	VAR robtarget Openhole_6902 := [[456.45, -15.03, 181.27], [0.011887, 0.707007, 0.706156, -0.036651], [0,0,0,0], [9E9, 9E9, 9E9, 9E9, 9E9, 9E9]];
	VAR robtarget Openhole_6903 := [[454.01, -15.03, 181.36], [0.00355, 0.707098, 0.706536, -0.028396], [0,0,0,0], [9E9, 9E9, 9E9, 9E9, 9E9, 9E9]];
	VAR robtarget Openhole_6904 := [[454.58, -16.45, 181.41], [0.010332, 0.707031, 0.706647, -0.025509], [0,0,0,0], [9E9, 9E9, 9E9, 9E9, 9E9, 9E9]];
	VAR robtarget Openhole_6905 := [[457.02, -16.45, 181.35], [0.018656, 0.706861, 0.7063, -0.033765], [0,0,0,0], [9E9, 9E9, 9E9, 9E9, 9E9, 9E9]];
	VAR robtarget Openhole_6906 := [[457.6, -16.2, 181.32], [0.019746, 0.706831, 0.706161, -0.036559], [0,0,0,0], [9E9, 9E9, 9E9, 9E9, 9E9, 9E9]];
	VAR robtarget Openhole_6907 := [[458.49, -15.74, 181.25], [0.021192, 0.706789, 0.705912, -0.041085], [0,0,0,0], [9E9, 9E9, 9E9, 9E9, 9E9, 9E9]];
	VAR robtarget Openhole_6908 := [[458.92, -15.49, 181.22], [0.021819, 0.70677, 0.705775, -0.043372], [0,0,0,0], [9E9, 9E9, 9E9, 9E9, 9E9, 9E9]];
	VAR robtarget Openhole_6909 := [[459.34, -15.23, 181.18], [0.022372, 0.706753, 0.70563, -0.045673], [0,0,0,0], [9E9, 9E9, 9E9, 9E9, 9E9, 9E9]];
	VAR robtarget Openhole_6910 := [[460.18, -14.69, 181.09], [0.023376, 0.70672, 0.705316, -0.050289], [0,0,0,0], [9E9, 9E9, 9E9, 9E9, 9E9, 9E9]];
	VAR robtarget Openhole_6911 := [[461.04, -14.18, 181], [0.024553, 0.70668, 0.704976, -0.05485], [0,0,0,0], [9E9, 9E9, 9E9, 9E9, 9E9, 9E9]];
	VAR robtarget Openhole_6912 := [[463.23, -13.02, 180.74], [0.028061, 0.70655, 0.704018, -0.066023], [0,0,0,0], [9E9, 9E9, 9E9, 9E9, 9E9, 9E9]];
	VAR robtarget Openhole_6913 := [[463.68, -12.81, 180.68], [0.028865, 0.706517, 0.703809, -0.068211], [0,0,0,0], [9E9, 9E9, 9E9, 9E9, 9E9, 9E9]];
	VAR robtarget Openhole_6914 := [[465.05, -12.22, 180.51], [0.031491, 0.706405, 0.703154, -0.074666], [0,0,0,0], [9E9, 9E9, 9E9, 9E9, 9E9, 9E9]];
	VAR robtarget Openhole_6915 := [[465.52, -12.04, 180.45], [0.032438, 0.706362, 0.702926, -0.076778], [0,0,0,0], [9E9, 9E9, 9E9, 9E9, 9E9, 9E9]];
	VAR robtarget Openhole_6916 := [[468.83, -10.99, 180.03], [0.040018, 0.705973, 0.701231, -0.090969], [0,0,0,0], [9E9, 9E9, 9E9, 9E9, 9E9, 9E9]];
	VAR robtarget Openhole_6917 := [[469.79, -10.75, 179.91], [0.042431, 0.705833, 0.700718, -0.094841], [0,0,0,0], [9E9, 9E9, 9E9, 9E9, 9E9, 9E9]];
	VAR robtarget Openhole_6918 := [[473.7, -10.06, 179.44], [0.053059, 0.705113, 0.698584, -0.109453], [0,0,0,0], [9E9, 9E9, 9E9, 9E9, 9E9, 9E9]];
	VAR robtarget Openhole_6919 := [[478.16, -9.69, 178.95], [0.066329, 0.703989, 0.69608, -0.124391], [0,0,0,0], [9E9, 9E9, 9E9, 9E9, 9E9, 9E9]];
	VAR robtarget Openhole_6920 := [[482.14, -9.61, 178.57], [0.078785, 0.702704, 0.693795, -0.136561], [0,0,0,0], [9E9, 9E9, 9E9, 9E9, 9E9, 9E9]];
	VAR robtarget Openhole_6921 := [[482.64, -9.62, 178.53], [0.080362, 0.702525, 0.693505, -0.138025], [0,0,0,0], [9E9, 9E9, 9E9, 9E9, 9E9, 9E9]];
	VAR robtarget Openhole_6922 := [[494.1, -10.02, 177.66], [0.116451, 0.697452, 0.686579, -0.169145], [0,0,0,0], [9E9, 9E9, 9E9, 9E9, 9E9, 9E9]];
	VAR robtarget Openhole_6923 := [[499.58, -10.13, 177.24], [0.132483, 0.694585, 0.682946, -0.183261], [0,0,0,0], [9E9, 9E9, 9E9, 9E9, 9E9, 9E9]];
	VAR robtarget Openhole_6924 := [[500.08, -10.12, 177.19], [0.13387, 0.694319, 0.6826, -0.184545], [0,0,0,0], [9E9, 9E9, 9E9, 9E9, 9E9, 9E9]];
	VAR robtarget Openhole_6925 := [[503.56, -10.02, 176.84], [0.143142, 0.692467, 0.680083, -0.193618], [0,0,0,0], [9E9, 9E9, 9E9, 9E9, 9E9, 9E9]];
	VAR robtarget Openhole_6926 := [[504.33, -10, 176.77], [0.145205, 0.692037, 0.679524, -0.19557], [0,0,0,0], [9E9, 9E9, 9E9, 9E9, 9E9, 9E9]];
	VAR robtarget Openhole_6927 := [[509.33, -10, 176.33], [0.183051, 0.683002, 0.683002, -0.183051], [0,0,0,0], [9E9, 9E9, 9E9, 9E9, 9E9, 9E9]];
	VAR robtarget Openhole_6928 := [[536.33, -10, 176.25], [0.183051, 0.683002, 0.683002, -0.183051], [0,0,0,0], [9E9, 9E9, 9E9, 9E9, 9E9, 9E9]];
	VAR robtarget Openhole_6929 := [[536.33, -10.89, 176.76], [0.183051, 0.683002, 0.683002, -0.183051], [0,0,0,0], [9E9, 9E9, 9E9, 9E9, 9E9, 9E9]];
	VAR robtarget Openhole_6930 := [[524.33, -10.89, 176.79], [0.183051, 0.683002, 0.683002, -0.183051], [0,0,0,0], [9E9, 9E9, 9E9, 9E9, 9E9, 9E9]];
	VAR robtarget Openhole_6931 := [[509.33, -10.89, 176.84], [0.183051, 0.683002, 0.683002, -0.183051], [0,0,0,0], [9E9, 9E9, 9E9, 9E9, 9E9, 9E9]];
	VAR robtarget Openhole_6932 := [[504.39, -10.89, 177.23], [0.147958, 0.691454, 0.680206, -0.193184], [0,0,0,0], [9E9, 9E9, 9E9, 9E9, 9E9, 9E9]];
	VAR robtarget Openhole_6933 := [[498.87, -11.14, 177.78], [0.133522, 0.694386, 0.684219, -0.178448], [0,0,0,0], [9E9, 9E9, 9E9, 9E9, 9E9, 9E9]];
	VAR robtarget Openhole_6934 := [[497.37, -11.14, 177.9], [0.129323, 0.69518, 0.685234, -0.17451], [0,0,0,0], [9E9, 9E9, 9E9, 9E9, 9E9, 9E9]];
	VAR robtarget Openhole_6935 := [[496.87, -11.14, 177.93], [0.127897, 0.695444, 0.685566, -0.173201], [0,0,0,0], [9E9, 9E9, 9E9, 9E9, 9E9, 9E9]];
	VAR robtarget Openhole_6936 := [[482.41, -10.79, 178.92], [0.083436, 0.702167, 0.694362, -0.133645], [0,0,0,0], [9E9, 9E9, 9E9, 9E9, 9E9, 9E9]];
	VAR robtarget Openhole_6937 := [[481.91, -10.8, 178.96], [0.081871, 0.702351, 0.694646, -0.132162], [0,0,0,0], [9E9, 9E9, 9E9, 9E9, 9E9, 9E9]];
	VAR robtarget Openhole_6938 := [[476.44, -10.97, 179.44], [0.064947, 0.704118, 0.697689, -0.115023], [0,0,0,0], [9E9, 9E9, 9E9, 9E9, 9E9, 9E9]];
	VAR robtarget Openhole_6939 := [[472.49, -11.44, 179.85], [0.053603, 0.705072, 0.699831, -0.101179], [0,0,0,0], [9E9, 9E9, 9E9, 9E9, 9E9, 9E9]];
	VAR robtarget Openhole_6940 := [[471.02, -11.7, 180.01], [0.049631, 0.705363, 0.700605, -0.09567], [0,0,0,0], [9E9, 9E9, 9E9, 9E9, 9E9, 9E9]];
	VAR robtarget Openhole_6941 := [[470.53, -11.8, 180.07], [0.048363, 0.705451, 0.70086, -0.093784], [0,0,0,0], [9E9, 9E9, 9E9, 9E9, 9E9, 9E9]];
	VAR robtarget Openhole_6942 := [[469.57, -12.03, 180.18], [0.045918, 0.705614, 0.701364, -0.089939], [0,0,0,0], [9E9, 9E9, 9E9, 9E9, 9E9, 9E9]];
	VAR robtarget Openhole_6943 := [[468.61, -12.29, 180.29], [0.043599, 0.705761, 0.701858, -0.085997], [0,0,0,0], [9E9, 9E9, 9E9, 9E9, 9E9, 9E9]];
	VAR robtarget Openhole_6944 := [[467.66, -12.58, 180.4], [0.041406, 0.705893, 0.70234, -0.081965], [0,0,0,0], [9E9, 9E9, 9E9, 9E9, 9E9, 9E9]];
	VAR robtarget Openhole_6945 := [[466.25, -13.07, 180.57], [0.038376, 0.706065, 0.703038, -0.075748], [0,0,0,0], [9E9, 9E9, 9E9, 9E9, 9E9, 9E9]];
	VAR robtarget Openhole_6946 := [[465.79, -13.26, 180.63], [0.037449, 0.706114, 0.703263, -0.073629], [0,0,0,0], [9E9, 9E9, 9E9, 9E9, 9E9, 9E9]];
	VAR robtarget Openhole_6947 := [[465.33, -13.45, 180.68], [0.036568, 0.706161, 0.703484, -0.071485], [0,0,0,0], [9E9, 9E9, 9E9, 9E9, 9E9, 9E9]];
	VAR robtarget Openhole_6948 := [[464.88, -13.66, 180.74], [0.035745, 0.706203, 0.703701, -0.069315], [0,0,0,0], [9E9, 9E9, 9E9, 9E9, 9E9, 9E9]];
	VAR robtarget Openhole_6949 := [[463.11, -14.56, 180.95], [0.032844, 0.706344, 0.704518, -0.060455], [0,0,0,0], [9E9, 9E9, 9E9, 9E9, 9E9, 9E9]];
	VAR robtarget Openhole_6950 := [[461.82, -15.31, 181.1], [0.031032, 0.706426, 0.705068, -0.053658], [0,0,0,0], [9E9, 9E9, 9E9, 9E9, 9E9, 9E9]];
	VAR robtarget Openhole_6951 := [[460.15, -16.4, 181.27], [0.029071, 0.706509, 0.705709, -0.044434], [0,0,0,0], [9E9, 9E9, 9E9, 9E9, 9E9, 9E9]];
	VAR robtarget Openhole_6952 := [[459.72, -16.65, 181.3], [0.028476, 0.706533, 0.70585, -0.042143], [0,0,0,0], [9E9, 9E9, 9E9, 9E9, 9E9, 9E9]];
	VAR robtarget Openhole_6953 := [[459.27, -16.88, 181.34], [0.027718, 0.706563, 0.70598, -0.039897], [0,0,0,0], [9E9, 9E9, 9E9, 9E9, 9E9, 9E9]];
	VAR robtarget Openhole_6954 := [[458.82, -17.08, 181.36], [0.026869, 0.706596, 0.706102, -0.037679], [0,0,0,0], [9E9, 9E9, 9E9, 9E9, 9E9, 9E9]];
	VAR robtarget Openhole_6955 := [[458.35, -17.26, 181.39], [0.025912, 0.706632, 0.706215, -0.035503], [0,0,0,0], [9E9, 9E9, 9E9, 9E9, 9E9, 9E9]];
	VAR robtarget Openhole_6956 := [[457.88, -17.43, 181.41], [0.024897, 0.706668, 0.70632, -0.033349], [0,0,0,0], [9E9, 9E9, 9E9, 9E9, 9E9, 9E9]];
	VAR robtarget Openhole_6957 := [[457.27, -17.6, 181.43], [0.023386, 0.70672, 0.706439, -0.030721], [0,0,0,0], [9E9, 9E9, 9E9, 9E9, 9E9, 9E9]];
	VAR robtarget Openhole_6958 := [[454.82, -17.6, 181.47], [0.015072, 0.706946, 0.70675, -0.02246], [0,0,0,0], [9E9, 9E9, 9E9, 9E9, 9E9, 9E9]];
	VAR robtarget Openhole_6959 := [[454.9, -18.58, 181.52], [0.018658, 0.706861, 0.70684, -0.019405], [0,0,0,0], [9E9, 9E9, 9E9, 9E9, 9E9, 9E9]];
	VAR robtarget Openhole_6960 := [[457.35, -18.58, 181.51], [0.026965, 0.706592, 0.706565, -0.027672], [0,0,0,0], [9E9, 9E9, 9E9, 9E9, 9E9, 9E9]];
	VAR robtarget Openhole_6961 := [[457.46, -18.57, 181.51], [0.027362, 0.706577, 0.706549, -0.028077], [0,0,0,0], [9E9, 9E9, 9E9, 9E9, 9E9, 9E9]];
	VAR robtarget Openhole_6962 := [[457.96, -18.57, 181.5], [0.029039, 0.70651, 0.70648, -0.029777], [0,0,0,0], [9E9, 9E9, 9E9, 9E9, 9E9, 9E9]];
	VAR robtarget Openhole_6963 := [[458.45, -18.46, 181.49], [0.030319, 0.706456, 0.706392, -0.031788], [0,0,0,0], [9E9, 9E9, 9E9, 9E9, 9E9, 9E9]];
	VAR robtarget Openhole_6964 := [[459.42, -18.22, 181.46], [0.032768, 0.706347, 0.706196, -0.03587], [0,0,0,0], [9E9, 9E9, 9E9, 9E9, 9E9, 9E9]];
	VAR robtarget Openhole_6965 := [[460.38, -17.92, 181.42], [0.034974, 0.706241, 0.70597, -0.040073], [0,0,0,0], [9E9, 9E9, 9E9, 9E9, 9E9, 9E9]];
	VAR robtarget Openhole_6966 := [[460.84, -17.74, 181.4], [0.035928, 0.706193, 0.705844, -0.042242], [0,0,0,0], [9E9, 9E9, 9E9, 9E9, 9E9, 9E9]];
	VAR robtarget Openhole_6967 := [[461.3, -17.54, 181.37], [0.036825, 0.706147, 0.70571, -0.044431], [0,0,0,0], [9E9, 9E9, 9E9, 9E9, 9E9, 9E9]];
	VAR robtarget Openhole_6968 := [[462.19, -17.09, 181.3], [0.038265, 0.706071, 0.705412, -0.048924], [0,0,0,0], [9E9, 9E9, 9E9, 9E9, 9E9, 9E9]];
	VAR robtarget Openhole_6969 := [[463.94, -16.14, 181.14], [0.040966, 0.705919, 0.704731, -0.057919], [0,0,0,0], [9E9, 9E9, 9E9, 9E9, 9E9, 9E9]];
	VAR robtarget Openhole_6970 := [[464.83, -15.7, 181.05], [0.042438, 0.705832, 0.704352, -0.062353], [0,0,0,0], [9E9, 9E9, 9E9, 9E9, 9E9, 9E9]];
	VAR robtarget Openhole_6971 := [[465.74, -15.28, 180.95], [0.044037, 0.705734, 0.703952, -0.066725], [0,0,0,0], [9E9, 9E9, 9E9, 9E9, 9E9, 9E9]];
	VAR robtarget Openhole_6972 := [[466.19, -15.08, 180.9], [0.044895, 0.70568, 0.703744, -0.068883], [0,0,0,0], [9E9, 9E9, 9E9, 9E9, 9E9, 9E9]];
	VAR robtarget Openhole_6973 := [[466.65, -14.89, 180.85], [0.045793, 0.705622, 0.703531, -0.071019], [0,0,0,0], [9E9, 9E9, 9E9, 9E9, 9E9, 9E9]];
	VAR robtarget Openhole_6974 := [[467.12, -14.71, 180.8], [0.046745, 0.70556, 0.703315, -0.073127], [0,0,0,0], [9E9, 9E9, 9E9, 9E9, 9E9, 9E9]];
	VAR robtarget Openhole_6975 := [[467.59, -14.54, 180.75], [0.047745, 0.705493, 0.703096, -0.075209], [0,0,0,0], [9E9, 9E9, 9E9, 9E9, 9E9, 9E9]];
	VAR robtarget Openhole_6976 := [[468.53, -14.24, 180.66], [0.049866, 0.705346, 0.702646, -0.079298], [0,0,0,0], [9E9, 9E9, 9E9, 9E9, 9E9, 9E9]];
	VAR robtarget Openhole_6977 := [[469.49, -13.97, 180.56], [0.052134, 0.705182, 0.702185, -0.083288], [0,0,0,0], [9E9, 9E9, 9E9, 9E9, 9E9, 9E9]];
	VAR robtarget Openhole_6978 := [[470.46, -13.73, 180.46], [0.054514, 0.705002, 0.701711, -0.087191], [0,0,0,0], [9E9, 9E9, 9E9, 9E9, 9E9, 9E9]];
	VAR robtarget Openhole_6979 := [[470.94, -13.62, 180.42], [0.055746, 0.704906, 0.70147, -0.089109], [0,0,0,0], [9E9, 9E9, 9E9, 9E9, 9E9, 9E9]];
	VAR robtarget Openhole_6980 := [[471.92, -13.42, 180.32], [0.058297, 0.7047, 0.700981, -0.092871], [0,0,0,0], [9E9, 9E9, 9E9, 9E9, 9E9, 9E9]];
	VAR robtarget Openhole_6981 := [[475.87, -12.91, 179.98], [0.069482, 0.703685, 0.69897, -0.106962], [0,0,0,0], [9E9, 9E9, 9E9, 9E9, 9E9, 9E9]];
	VAR robtarget Openhole_6982 := [[480.85, -12.71, 179.63], [0.084707, 0.702015, 0.696348, -0.122882], [0,0,0,0], [9E9, 9E9, 9E9, 9E9, 9E9, 9E9]];
	VAR robtarget Openhole_6983 := [[482.35, -12.7, 179.53], [0.089365, 0.701437, 0.695534, -0.127408], [0,0,0,0], [9E9, 9E9, 9E9, 9E9, 9E9, 9E9]];
	VAR robtarget Openhole_6984 := [[482.85, -12.7, 179.5], [0.090921, 0.701237, 0.69526, -0.128895], [0,0,0,0], [9E9, 9E9, 9E9, 9E9, 9E9, 9E9]];
	VAR robtarget Openhole_6985 := [[495.33, -12.89, 178.83], [0.12882, 0.695274, 0.687872, -0.163806], [0,0,0,0], [9E9, 9E9, 9E9, 9E9, 9E9, 9E9]];
	VAR robtarget Openhole_6986 := [[495.83, -12.89, 178.8], [0.130242, 0.695009, 0.687549, -0.165156], [0,0,0,0], [9E9, 9E9, 9E9, 9E9, 9E9, 9E9]];
	VAR robtarget Openhole_6987 := [[501.81, -12.75, 178.37], [0.146466, 0.691771, 0.683473, -0.181287], [0,0,0,0], [9E9, 9E9, 9E9, 9E9, 9E9, 9E9]];
	VAR robtarget Openhole_6988 := [[504.34, -12.58, 178.13], [0.152777, 0.690405, 0.681616, -0.188149], [0,0,0,0], [9E9, 9E9, 9E9, 9E9, 9E9, 9E9]];
	VAR robtarget Openhole_6989 := [[509.34, -12.58, 177.82], [0.183051, 0.683002, 0.683002, -0.183051], [0,0,0,0], [9E9, 9E9, 9E9, 9E9, 9E9, 9E9]];
	VAR robtarget Openhole_6990 := [[536.34, -12.58, 177.74], [0.183051, 0.683002, 0.683002, -0.183051], [0,0,0,0], [9E9, 9E9, 9E9, 9E9, 9E9, 9E9]];
	VAR robtarget Openhole_6991 := [[536.34, -16.49, 179.99], [0.183051, 0.683002, 0.683002, -0.183051], [0,0,0,0], [9E9, 9E9, 9E9, 9E9, 9E9, 9E9]];
	VAR robtarget Openhole_6992 := [[509.34, -16.49, 180.08], [0.183051, 0.683002, 0.683002, -0.183051], [0,0,0,0], [9E9, 9E9, 9E9, 9E9, 9E9, 9E9]];
	VAR robtarget Openhole_6993 := [[504.34, -16.49, 180.2], [0.164245, 0.687767, 0.684639, -0.176832], [0,0,0,0], [9E9, 9E9, 9E9, 9E9, 9E9, 9E9]];
	VAR robtarget Openhole_6994 := [[497.74, -16.81, 180.51], [0.147487, 0.691555, 0.6891, -0.158559], [0,0,0,0], [9E9, 9E9, 9E9, 9E9, 9E9, 9E9]];
	VAR robtarget Openhole_6995 := [[491.75, -16.89, 180.67], [0.130825, 0.694899, 0.692766, -0.141687], [0,0,0,0], [9E9, 9E9, 9E9, 9E9, 9E9, 9E9]];
	VAR robtarget Openhole_6996 := [[491.25, -16.89, 180.68], [0.129379, 0.69517, 0.693055, -0.140267], [0,0,0,0], [9E9, 9E9, 9E9, 9E9, 9E9, 9E9]];
	VAR robtarget Openhole_6997 := [[478.25, -16.73, 180.9], [0.089551, 0.701413, 0.699715, -0.101979], [0,0,0,0], [9E9, 9E9, 9E9, 9E9, 9E9, 9E9]];
	VAR robtarget Openhole_6998 := [[477.75, -16.74, 180.92], [0.087979, 0.701612, 0.69994, -0.100419], [0,0,0,0], [9E9, 9E9, 9E9, 9E9, 9E9, 9E9]];
	VAR robtarget Openhole_6999 := [[472.25, -16.88, 181.07], [0.070842, 0.703549, 0.702268, -0.082577], [0,0,0,0], [9E9, 9E9, 9E9, 9E9, 9E9, 9E9]];
	VAR robtarget Openhole_7000 := [[471.26, -16.95, 181.1], [0.067854, 0.703844, 0.702666, -0.079124], [0,0,0,0], [9E9, 9E9, 9E9, 9E9, 9E9, 9E9]];
	VAR robtarget Openhole_7001 := [[470.26, -17.06, 181.15], [0.064977, 0.704115, 0.703059, -0.075554], [0,0,0,0], [9E9, 9E9, 9E9, 9E9, 9E9, 9E9]];
	VAR robtarget Openhole_7002 := [[468.29, -17.35, 181.24], [0.059459, 0.704602, 0.703814, -0.068163], [0,0,0,0], [9E9, 9E9, 9E9, 9E9, 9E9, 9E9]];
	VAR robtarget Openhole_7003 := [[467.8, -17.44, 181.26], [0.058137, 0.704713, 0.703995, -0.06626], [0,0,0,0], [9E9, 9E9, 9E9, 9E9, 9E9, 9E9]];
	VAR robtarget Openhole_7004 := [[467.31, -17.54, 181.28], [0.056855, 0.704817, 0.704175, -0.064325], [0,0,0,0], [9E9, 9E9, 9E9, 9E9, 9E9, 9E9]];
	VAR robtarget Openhole_7005 := [[465.37, -18.02, 181.39], [0.052018, 0.705191, 0.704858, -0.056353], [0,0,0,0], [9E9, 9E9, 9E9, 9E9, 9E9, 9E9]];
	VAR robtarget Openhole_7006 := [[464.4, -18.28, 181.43], [0.049714, 0.705357, 0.705172, -0.052273], [0,0,0,0], [9E9, 9E9, 9E9, 9E9, 9E9, 9E9]];
	VAR robtarget Openhole_7007 := [[463.44, -18.53, 181.47], [0.047307, 0.705523, 0.70546, -0.048235], [0,0,0,0], [9E9, 9E9, 9E9, 9E9, 9E9, 9E9]];
	VAR robtarget Openhole_7008 := [[460.01, -19.25, 181.56], [0.03826, 0.706071, 0.706271, -0.034365], [0,0,0,0], [9E9, 9E9, 9E9, 9E9, 9E9, 9E9]];
	VAR robtarget Openhole_7009 := [[458.04, -19.56, 181.59], [0.032644, 0.706353, 0.706604, -0.026672], [0,0,0,0], [9E9, 9E9, 9E9, 9E9, 9E9, 9E9]];
	VAR robtarget Openhole_7010 := [[457.3, -19.61, 181.59], [0.03031, 0.706457, 0.706699, -0.024], [0,0,0,0], [9E9, 9E9, 9E9, 9E9, 9E9, 9E9]];
	VAR robtarget Openhole_7011 := [[454.85, -19.61, 181.57], [0.022009, 0.706764, 0.706932, -0.015726], [0,0,0,0], [9E9, 9E9, 9E9, 9E9, 9E9, 9E9]];
	VAR robtarget Openhole_7012 := [[454.66, -20.66, 181.62], [0.024932, 0.706667, 0.707013, -0.011519], [0,0,0,0], [9E9, 9E9, 9E9, 9E9, 9E9, 9E9]];
	VAR robtarget Openhole_7013 := [[457.1, -20.66, 181.66], [0.033229, 0.706326, 0.706829, -0.019801], [0,0,0,0], [9E9, 9E9, 9E9, 9E9, 9E9, 9E9]];
	VAR robtarget Openhole_7014 := [[457.65, -20.63, 181.67], [0.034967, 0.706242, 0.706773, -0.021725], [0,0,0,0], [9E9, 9E9, 9E9, 9E9, 9E9, 9E9]];
	VAR robtarget Openhole_7015 := [[458.63, -20.47, 181.67], [0.037739, 0.706099, 0.706643, -0.025609], [0,0,0,0], [9E9, 9E9, 9E9, 9E9, 9E9, 9E9]];
	VAR robtarget Openhole_7016 := [[459.13, -20.43, 181.67], [0.039281, 0.706015, 0.706575, -0.027426], [0,0,0,0], [9E9, 9E9, 9E9, 9E9, 9E9, 9E9]];
	VAR robtarget Openhole_7017 := [[460.13, -20.37, 181.68], [0.042453, 0.705831, 0.706428, -0.030973], [0,0,0,0], [9E9, 9E9, 9E9, 9E9, 9E9, 9E9]];
	VAR robtarget Openhole_7018 := [[461.63, -20.35, 181.7], [0.047407, 0.705516, 0.706186, -0.036083], [0,0,0,0], [9E9, 9E9, 9E9, 9E9, 9E9, 9E9]];
	VAR robtarget Openhole_7019 := [[462.63, -20.37, 181.71], [0.050804, 0.705279, 0.70601, -0.039375], [0,0,0,0], [9E9, 9E9, 9E9, 9E9, 9E9, 9E9]];
	VAR robtarget Openhole_7020 := [[464.13, -20.42, 181.74], [0.055995, 0.704886, 0.705726, -0.044175], [0,0,0,0], [9E9, 9E9, 9E9, 9E9, 9E9, 9E9]];
	VAR robtarget Openhole_7021 := [[480.61, -20.9, 182.11], [0.11041, 0.698434, 0.700578, -0.095867], [0,0,0,0], [9E9, 9E9, 9E9, 9E9, 9E9, 9E9]];
	VAR robtarget Openhole_7022 := [[489.11, -20.98, 182.29], [0.135964, 0.693912, 0.696615, -0.121355], [0,0,0,0], [9E9, 9E9, 9E9, 9E9, 9E9, 9E9]];
	VAR robtarget Openhole_7023 := [[489.61, -20.98, 182.3], [0.137402, 0.693629, 0.696357, -0.122828], [0,0,0,0], [9E9, 9E9, 9E9, 9E9, 9E9, 9E9]];
	VAR robtarget Openhole_7024 := [[499.61, -20.8, 182.4], [0.164519, 0.687702, 0.690652, -0.151655], [0,0,0,0], [9E9, 9E9, 9E9, 9E9, 9E9, 9E9]];
	VAR robtarget Openhole_7025 := [[504.35, -20.6, 182.37], [0.176239, 0.684792, 0.687612, -0.164894], [0,0,0,0], [9E9, 9E9, 9E9, 9E9, 9E9, 9E9]];
	VAR robtarget Openhole_7026 := [[509.35, -20.6, 182.45], [0.183051, 0.683002, 0.683002, -0.183051], [0,0,0,0], [9E9, 9E9, 9E9, 9E9, 9E9, 9E9]];
	VAR robtarget Openhole_7027 := [[536.35, -20.6, 182.36], [0.183051, 0.683002, 0.683002, -0.183051], [0,0,0,0], [9E9, 9E9, 9E9, 9E9, 9E9, 9E9]];
	VAR robtarget Openhole_7028 := [[536.35, -22.17, 183.27], [0.183051, 0.683002, 0.683002, -0.183051], [0,0,0,0], [9E9, 9E9, 9E9, 9E9, 9E9, 9E9]];
	VAR robtarget Openhole_7029 := [[509.35, -22.17, 183.36], [0.183051, 0.683002, 0.683002, -0.183051], [0,0,0,0], [9E9, 9E9, 9E9, 9E9, 9E9, 9E9]];
	VAR robtarget Openhole_7030 := [[504.35, -22.17, 183.2], [0.180823, 0.683596, 0.688696, -0.160305], [0,0,0,0], [9E9, 9E9, 9E9, 9E9, 9E9, 9E9]];
	VAR robtarget Openhole_7031 := [[494.58, -22.52, 183.06], [0.156112, 0.689659, 0.694592, -0.132445], [0,0,0,0], [9E9, 9E9, 9E9, 9E9, 9E9, 9E9]];
	VAR robtarget Openhole_7032 := [[485.58, -22.61, 182.79], [0.130782, 0.694907, 0.699165, -0.105679], [0,0,0,0], [9E9, 9E9, 9E9, 9E9, 9E9, 9E9]];
	VAR robtarget Openhole_7033 := [[485.08, -22.61, 182.77], [0.129309, 0.695183, 0.699393, -0.10416], [0,0,0,0], [9E9, 9E9, 9E9, 9E9, 9E9, 9E9]];
	VAR robtarget Openhole_7034 := [[471.6, -22.42, 182.27], [0.08706, 0.701727, 0.704369, -0.06216], [0,0,0,0], [9E9, 9E9, 9E9, 9E9, 9E9, 9E9]];
	VAR robtarget Openhole_7035 := [[465.61, -22.1, 182.02], [0.066522, 0.703971, 0.705767, -0.043507], [0,0,0,0], [9E9, 9E9, 9E9, 9E9, 9E9, 9E9]];
	VAR robtarget Openhole_7036 := [[461.64, -21.66, 181.85], [0.051867, 0.705202, 0.706396, -0.031702], [0,0,0,0], [9E9, 9E9, 9E9, 9E9, 9E9, 9E9]];
	VAR robtarget Openhole_7037 := [[460.14, -21.53, 181.8], [0.046434, 0.705581, 0.706587, -0.027111], [0,0,0,0], [9E9, 9E9, 9E9, 9E9, 9E9, 9E9]];
	VAR robtarget Openhole_7038 := [[459.65, -21.51, 181.79], [0.044669, 0.705694, 0.706646, -0.025518], [0,0,0,0], [9E9, 9E9, 9E9, 9E9, 9E9, 9E9]];
	VAR robtarget Openhole_7039 := [[459.15, -21.49, 181.77], [0.042948, 0.705801, 0.706704, -0.023876], [0,0,0,0], [9E9, 9E9, 9E9, 9E9, 9E9, 9E9]];
	VAR robtarget Openhole_7040 := [[458.65, -21.5, 181.76], [0.041268, 0.705902, 0.706759, -0.022186], [0,0,0,0], [9E9, 9E9, 9E9, 9E9, 9E9, 9E9]];
	VAR robtarget Openhole_7041 := [[458.15, -21.51, 181.75], [0.039639, 0.705995, 0.706811, -0.020445], [0,0,0,0], [9E9, 9E9, 9E9, 9E9, 9E9, 9E9]];
	VAR robtarget Openhole_7042 := [[457.66, -21.63, 181.75], [0.038399, 0.706063, 0.706867, -0.018405], [0,0,0,0], [9E9, 9E9, 9E9, 9E9, 9E9, 9E9]];
	VAR robtarget Openhole_7043 := [[456.8, -21.6, 181.73], [0.035413, 0.706219, 0.706935, -0.01559], [0,0,0,0], [9E9, 9E9, 9E9, 9E9, 9E9, 9E9]];
	VAR robtarget Openhole_7044 := [[454.35, -21.6, 181.67], [0.027119, 0.706587, 0.707069, -0.0073], [0,0,0,0], [9E9, 9E9, 9E9, 9E9, 9E9, 9E9]];
	VAR robtarget Openhole_7045 := [[453.91, -22.56, 181.7], [0.028848, 0.706518, 0.707102, -0.002564], [0,0,0,0], [9E9, 9E9, 9E9, 9E9, 9E9, 9E9]];
	VAR robtarget Openhole_7046 := [[456.36, -22.56, 181.78], [0.037142, 0.706131, 0.707023, -0.010862], [0,0,0,0], [9E9, 9E9, 9E9, 9E9, 9E9, 9E9]];
	VAR robtarget Openhole_7047 := [[456.89, -22.57, 181.8], [0.039015, 0.70603, 0.706994, -0.012629], [0,0,0,0], [9E9, 9E9, 9E9, 9E9, 9E9, 9E9]];
	VAR robtarget Openhole_7048 := [[457.39, -22.58, 181.82], [0.040716, 0.705934, 0.706962, -0.014306], [0,0,0,0], [9E9, 9E9, 9E9, 9E9, 9E9, 9E9]];
	VAR robtarget Openhole_7049 := [[458.89, -22.62, 181.87], [0.045917, 0.705614, 0.706846, -0.019217], [0,0,0,0], [9E9, 9E9, 9E9, 9E9, 9E9, 9E9]];
	VAR robtarget Openhole_7050 := [[459.89, -22.67, 181.91], [0.049444, 0.705376, 0.706752, -0.022408], [0,0,0,0], [9E9, 9E9, 9E9, 9E9, 9E9, 9E9]];
	VAR robtarget Openhole_7051 := [[465.84, -23.34, 182.23], [0.071439, 0.703489, 0.705966, -0.040151], [0,0,0,0], [9E9, 9E9, 9E9, 9E9, 9E9, 9E9]];
	VAR robtarget Openhole_7052 := [[472.83, -23.6, 182.58], [0.094896, 0.70071, 0.704358, -0.062286], [0,0,0,0], [9E9, 9E9, 9E9, 9E9, 9E9, 9E9]];
	VAR robtarget Openhole_7053 := [[480.32, -23.66, 182.92], [0.11838, 0.697127, 0.701849, -0.086071], [0,0,0,0], [9E9, 9E9, 9E9, 9E9, 9E9, 9E9]];
	VAR robtarget Openhole_7054 := [[480.82, -23.66, 182.94], [0.119895, 0.696868, 0.701655, -0.087638], [0,0,0,0], [9E9, 9E9, 9E9, 9E9, 9E9, 9E9]];
	VAR robtarget Openhole_7055 := [[481.32, -23.66, 182.97], [0.121406, 0.696606, 0.701458, -0.089201], [0,0,0,0], [9E9, 9E9, 9E9, 9E9, 9E9, 9E9]];
	VAR robtarget Openhole_7056 := [[481.82, -23.66, 182.99], [0.122908, 0.696343, 0.701258, -0.090763], [0,0,0,0], [9E9, 9E9, 9E9, 9E9, 9E9, 9E9]];
	VAR robtarget Openhole_7057 := [[495.81, -23.48, 183.53], [0.162364, 0.688214, 0.694482, -0.133023], [0,0,0,0], [9E9, 9E9, 9E9, 9E9, 9E9, 9E9]];
	VAR robtarget Openhole_7058 := [[504.35, -23.14, 183.72], [0.183639, 0.682845, 0.689348, -0.157477], [0,0,0,0], [9E9, 9E9, 9E9, 9E9, 9E9, 9E9]];
	VAR robtarget Openhole_7059 := [[509.35, -23.14, 183.92], [0.183051, 0.683002, 0.683002, -0.183051], [0,0,0,0], [9E9, 9E9, 9E9, 9E9, 9E9, 9E9]];
	VAR robtarget Openhole_7060 := [[536.35, -23.14, 183.83], [0.183051, 0.683002, 0.683002, -0.183051], [0,0,0,0], [9E9, 9E9, 9E9, 9E9, 9E9, 9E9]];
	VAR robtarget Openhole_7061 := [[536.36, -24.03, 184.35], [0.183051, 0.683002, 0.683002, -0.183051], [0,0,0,0], [9E9, 9E9, 9E9, 9E9, 9E9, 9E9]];
	VAR robtarget Openhole_7062 := [[509.36, -24.03, 184.43], [0.183051, 0.683002, 0.683002, -0.183051], [0,0,0,0], [9E9, 9E9, 9E9, 9E9, 9E9, 9E9]];
	VAR robtarget Openhole_7063 := [[504.36, -24.03, 184.19], [0.186235, 0.682141, 0.68994, -0.154866], [0,0,0,0], [9E9, 9E9, 9E9, 9E9, 9E9, 9E9]];
	VAR robtarget Openhole_7064 := [[493.5, -24.43, 183.84], [0.158957, 0.689009, 0.69624, -0.123493], [0,0,0,0], [9E9, 9E9, 9E9, 9E9, 9E9, 9E9]];
	VAR robtarget Openhole_7065 := [[477.02, -24.66, 183.04], [0.111498, 0.698261, 0.703396, -0.072345], [0,0,0,0], [9E9, 9E9, 9E9, 9E9, 9E9, 9E9]];
	VAR robtarget Openhole_7066 := [[473.03, -24.68, 182.83], [0.099048, 0.700135, 0.704609, -0.059386], [0,0,0,0], [9E9, 9E9, 9E9, 9E9, 9E9, 9E9]];
	VAR robtarget Openhole_7067 := [[472.53, -24.68, 182.8], [0.097464, 0.700358, 0.704744, -0.057759], [0,0,0,0], [9E9, 9E9, 9E9, 9E9, 9E9, 9E9]];
	VAR robtarget Openhole_7068 := [[465.04, -24.53, 182.37], [0.072784, 0.703351, 0.706313, -0.033488], [0,0,0,0], [9E9, 9E9, 9E9, 9E9, 9E9, 9E9]];
	VAR robtarget Openhole_7069 := [[458.58, -23.97, 181.98], [0.049419, 0.705378, 0.706976, -0.013607], [0,0,0,0], [9E9, 9E9, 9E9, 9E9, 9E9, 9E9]];
	VAR robtarget Openhole_7070 := [[457.08, -23.91, 181.9], [0.044176, 0.705726, 0.707053, -0.008744], [0,0,0,0], [9E9, 9E9, 9E9, 9E9, 9E9, 9E9]];
	VAR robtarget Openhole_7071 := [[456.08, -23.86, 181.85], [0.040639, 0.705938, 0.707085, -0.005532], [0,0,0,0], [9E9, 9E9, 9E9, 9E9, 9E9, 9E9]];
	VAR robtarget Openhole_7072 := [[455.52, -23.79, 181.82], [0.038494, 0.706058, 0.707096, -0.003881], [0,0,0,0], [9E9, 9E9, 9E9, 9E9, 9E9, 9E9]];
	VAR robtarget Openhole_7073 := [[453.08, -23.79, 181.71], [0.030195, 0.706462, 0.707093, 0.004426], [0,0,0,0], [9E9, 9E9, 9E9, 9E9, 9E9, 9E9]];
	VAR robtarget Openhole_7074 := [[451.65, -25.14, 181.68], [0.02994, 0.706473, 0.706971, 0.013839], [0,0,0,0], [9E9, 9E9, 9E9, 9E9, 9E9, 9E9]];
	VAR robtarget Openhole_7075 := [[454.1, -25.14, 181.82], [0.038251, 0.706071, 0.707085, 0.005526], [0,0,0,0], [9E9, 9E9, 9E9, 9E9, 9E9, 9E9]];
	VAR robtarget Openhole_7076 := [[454.69, -25.32, 181.86], [0.040869, 0.705925, 0.707095, 0.00415], [0,0,0,0], [9E9, 9E9, 9E9, 9E9, 9E9, 9E9]];
	VAR robtarget Openhole_7077 := [[455.18, -25.38, 181.9], [0.042728, 0.705815, 0.707102, 0.002645], [0,0,0,0], [9E9, 9E9, 9E9, 9E9, 9E9, 9E9]];
	VAR robtarget Openhole_7078 := [[455.68, -25.42, 181.93], [0.044554, 0.705702, 0.707106, 0.001105], [0,0,0,0], [9E9, 9E9, 9E9, 9E9, 9E9, 9E9]];
	VAR robtarget Openhole_7079 := [[465.15, -25.83, 182.58], [0.077482, 0.702849, 0.706491, -0.029493], [0,0,0,0], [9E9, 9E9, 9E9, 9E9, 9E9, 9E9]];
	VAR robtarget Openhole_7080 := [[467.64, -25.85, 182.74], [0.085685, 0.701896, 0.706099, -0.037748], [0,0,0,0], [9E9, 9E9, 9E9, 9E9, 9E9, 9E9]];
	VAR robtarget Openhole_7081 := [[468.14, -25.85, 182.78], [0.087296, 0.701697, 0.706008, -0.039412], [0,0,0,0], [9E9, 9E9, 9E9, 9E9, 9E9, 9E9]];
	VAR robtarget Openhole_7082 := [[491.1, -25.41, 184.11], [0.155322, 0.689837, 0.697951, -0.113421], [0,0,0,0], [9E9, 9E9, 9E9, 9E9, 9E9, 9E9]];
	VAR robtarget Openhole_7083 := [[502.58, -25, 184.6], [0.184598, 0.682586, 0.691607, -0.147243], [0,0,0,0], [9E9, 9E9, 9E9, 9E9, 9E9, 9E9]];
	VAR robtarget Openhole_7084 := [[504.36, -24.92, 184.66], [0.188806, 0.681434, 0.690516, -0.152275], [0,0,0,0], [9E9, 9E9, 9E9, 9E9, 9E9, 9E9]];
	VAR robtarget Openhole_7085 := [[509.36, -24.92, 184.94], [0.183051, 0.683002, 0.683002, -0.183051], [0,0,0,0], [9E9, 9E9, 9E9, 9E9, 9E9, 9E9]];
	VAR robtarget Openhole_7086 := [[536.36, -24.92, 184.86], [0.183051, 0.683002, 0.683002, -0.183051], [0,0,0,0], [9E9, 9E9, 9E9, 9E9, 9E9, 9E9]];
	VAR robtarget Openhole_7087 := [[536.36, -25.98, 185.47], [0.183051, 0.683002, 0.683002, -0.183051], [0,0,0,0], [9E9, 9E9, 9E9, 9E9, 9E9, 9E9]];
	VAR robtarget Openhole_7088 := [[509.36, -25.98, 185.55], [0.183051, 0.683002, 0.683002, -0.183051], [0,0,0,0], [9E9, 9E9, 9E9, 9E9, 9E9, 9E9]];
	VAR robtarget Openhole_7089 := [[504.36, -25.98, 185.22], [0.191861, 0.68058, 0.691189, -0.149188], [0,0,0,0], [9E9, 9E9, 9E9, 9E9, 9E9, 9E9]];
	VAR robtarget Openhole_7090 := [[492.57, -26.46, 184.63], [0.162583, 0.688162, 0.697766, -0.114556], [0,0,0,0], [9E9, 9E9, 9E9, 9E9, 9E9, 9E9]];
	VAR robtarget Openhole_7091 := [[471.63, -27.19, 183.29], [0.102879, 0.699583, 0.705575, -0.046521], [0,0,0,0], [9E9, 9E9, 9E9, 9E9, 9E9, 9E9]];
	VAR robtarget Openhole_7092 := [[456.18, -27.73, 182.11], [0.05407, 0.705036, 0.70707, 0.007188], [0,0,0,0], [9E9, 9E9, 9E9, 9E9, 9E9, 9E9]];
	VAR robtarget Openhole_7093 := [[455.69, -27.74, 182.07], [0.052428, 0.705161, 0.707051, 0.008917], [0,0,0,0], [9E9, 9E9, 9E9, 9E9, 9E9, 9E9]];
	VAR robtarget Openhole_7094 := [[454.69, -27.73, 181.99], [0.049019, 0.705406, 0.707001, 0.012256], [0,0,0,0], [9E9, 9E9, 9E9, 9E9, 9E9, 9E9]];
	VAR robtarget Openhole_7095 := [[454.19, -27.71, 181.95], [0.047267, 0.705525, 0.706971, 0.013878], [0,0,0,0], [9E9, 9E9, 9E9, 9E9, 9E9, 9E9]];
	VAR robtarget Openhole_7096 := [[452.7, -27.62, 181.82], [0.041922, 0.705863, 0.706861, 0.018659], [0,0,0,0], [9E9, 9E9, 9E9, 9E9, 9E9, 9E9]];
	VAR robtarget Openhole_7097 := [[448.72, -27.39, 181.49], [0.027601, 0.706568, 0.70641, 0.031382], [0,0,0,0], [9E9, 9E9, 9E9, 9E9, 9E9, 9E9]];
	VAR robtarget Openhole_7098 := [[448.22, -27.39, 181.45], [0.025896, 0.706632, 0.706333, 0.033064], [0,0,0,0], [9E9, 9E9, 9E9, 9E9, 9E9, 9E9]];
	VAR robtarget Openhole_7099 := [[447.72, -27.4, 181.41], [0.024238, 0.706691, 0.70625, 0.034792], [0,0,0,0], [9E9, 9E9, 9E9, 9E9, 9E9, 9E9]];
	VAR robtarget Openhole_7100 := [[447.23, -27.43, 181.37], [0.022618, 0.706745, 0.706161, 0.036556], [0,0,0,0], [9E9, 9E9, 9E9, 9E9, 9E9, 9E9]];
	VAR robtarget Openhole_7101 := [[445.74, -27.57, 181.24], [0.018011, 0.706877, 0.705855, 0.042052], [0,0,0,0], [9E9, 9E9, 9E9, 9E9, 9E9, 9E9]];
	VAR robtarget Openhole_7102 := [[442.28, -28.03, 180.93], [0.007764, 0.707064, 0.704948, 0.05521], [0,0,0,0], [9E9, 9E9, 9E9, 9E9, 9E9, 9E9]];
	VAR robtarget Openhole_7103 := [[441.3, -28.17, 180.83], [0.004872, 0.70709, 0.704643, 0.058973], [0,0,0,0], [9E9, 9E9, 9E9, 9E9, 9E9, 9E9]];
	VAR robtarget Openhole_7104 := [[438.84, -28.58, 180.58], [-0.002114, 0.707104, 0.703781, 0.068497], [0,0,0,0], [9E9, 9E9, 9E9, 9E9, 9E9, 9E9]];
	VAR robtarget Openhole_7105 := [[437.87, -28.76, 180.47], [-0.004857, 0.70709, 0.703399, 0.072315], [0,0,0,0], [9E9, 9E9, 9E9, 9E9, 9E9, 9E9]];
	VAR robtarget Openhole_7106 := [[430.08, -30.27, 179.46], [-0.026214, 0.706621, 0.699631, 0.102548], [0,0,0,0], [9E9, 9E9, 9E9, 9E9, 9E9, 9E9]];
	VAR robtarget Openhole_7107 := [[425.17, -30.94, 178.77], [-0.040391, 0.705952, 0.696832, 0.120105], [0,0,0,0], [9E9, 9E9, 9E9, 9E9, 9E9, 9E9]];
	VAR robtarget Openhole_7108 := [[420.22, -31.24, 178.12], [-0.055673, 0.704912, 0.693884, 0.136105], [0,0,0,0], [9E9, 9E9, 9E9, 9E9, 9E9, 9E9]];
	VAR robtarget Openhole_7109 := [[418.24, -31.27, 177.88], [-0.06204, 0.70438, 0.692689, 0.142065], [0,0,0,0], [9E9, 9E9, 9E9, 9E9, 9E9, 9E9]];
	VAR robtarget Openhole_7110 := [[417.74, -31.27, 177.82], [-0.063646, 0.704237, 0.692389, 0.14352], [0,0,0,0], [9E9, 9E9, 9E9, 9E9, 9E9, 9E9]];
	VAR robtarget Openhole_7111 := [[411.78, -31.03, 177.2], [-0.083306, 0.702182, 0.688788, 0.159908], [0,0,0,0], [9E9, 9E9, 9E9, 9E9, 9E9, 9E9]];
	VAR robtarget Openhole_7112 := [[397.86, -29.96, 176.13], [-0.128027, 0.69542, 0.680085, 0.193607], [0,0,0,0], [9E9, 9E9, 9E9, 9E9, 9E9, 9E9]];
	VAR robtarget Openhole_7113 := [[394.33, -29.87, 175.8], [-0.138111, 0.693488, 0.677623, 0.202056], [0,0,0,0], [9E9, 9E9, 9E9, 9E9, 9E9, 9E9]];
	VAR robtarget Openhole_7114 := [[389.33, -29.87, 175.28], [-0.151564, 0.690672, 0.673997, 0.21384], [0,0,0,0], [9E9, 9E9, 9E9, 9E9, 9E9, 9E9]];
	VAR robtarget Openhole_7115 := [[362.33, -29.87, 175.36], [-0.183051, 0.683002, 0.683002, 0.183051], [0,0,0,0], [9E9, 9E9, 9E9, 9E9, 9E9, 9E9]];
	VAR robtarget Openhole_7116 := [[361.41, -38.7, 170.27], [-0.183051, 0.683002, 0.683002, 0.183051], [0,0,0,0], [9E9, 9E9, 9E9, 9E9, 9E9, 9E9]];
	VAR robtarget Openhole_7117 := [[389.31, -38.7, 170.18], [-0.126437, 0.695711, 0.665828, 0.23806], [0,0,0,0], [9E9, 9E9, 9E9, 9E9, 9E9, 9E9]];
	VAR robtarget Openhole_7118 := [[480.22, -38.7, 187.38], [0.165332, 0.687507, 0.706093, -0.037858], [0,0,0,0], [9E9, 9E9, 9E9, 9E9, 9E9, 9E9]];
	VAR robtarget Openhole_7119 := [[488.08, -37.66, 188.48], [0.184231, 0.682685, 0.703996, -0.066253], [0,0,0,0], [9E9, 9E9, 9E9, 9E9, 9E9, 9E9]];
	VAR robtarget Openhole_7120 := [[498.44, -36.73, 189.9], [0.208262, 0.675742, 0.699894, -0.100736], [0,0,0,0], [9E9, 9E9, 9E9, 9E9, 9E9, 9E9]];
	VAR robtarget Openhole_7121 := [[504.37, -36.35, 190.71], [0.221359, 0.671565, 0.697021, -0.119004], [0,0,0,0], [9E9, 9E9, 9E9, 9E9, 9E9, 9E9]];
	VAR robtarget Openhole_7122 := [[504.38, -36.35, 190.71], [0.221371, 0.671562, 0.697018, -0.119021], [0,0,0,0], [9E9, 9E9, 9E9, 9E9, 9E9, 9E9]];
	VAR robtarget Openhole_7123 := [[509.38, -36.35, 191.54], [0.183051, 0.683002, 0.683002, -0.183051], [0,0,0,0], [9E9, 9E9, 9E9, 9E9, 9E9, 9E9]];
	VAR robtarget Openhole_7124 := [[536.38, -36.35, 191.46], [0.183051, 0.683002, 0.683002, -0.183051], [0,0,0,0], [9E9, 9E9, 9E9, 9E9, 9E9, 9E9]];
	VAR robtarget Openhole_7125 := [[536.38, -35.46, 190.95], [0.183051, 0.683002, 0.683002, -0.183051], [0,0,0,0], [9E9, 9E9, 9E9, 9E9, 9E9, 9E9]];
	VAR robtarget Openhole_7126 := [[509.38, -35.46, 191.03], [0.183051, 0.683002, 0.683002, -0.183051], [0,0,0,0], [9E9, 9E9, 9E9, 9E9, 9E9, 9E9]];
	VAR robtarget Openhole_7127 := [[504.37, -35.46, 190.24], [0.218896, 0.672372, 0.696577, -0.121577], [0,0,0,0], [9E9, 9E9, 9E9, 9E9, 9E9, 9E9]];
	VAR robtarget Openhole_7128 := [[504.37, -35.46, 190.24], [0.218891, 0.672374, 0.696578, -0.12157], [0,0,0,0], [9E9, 9E9, 9E9, 9E9, 9E9, 9E9]];
	VAR robtarget Openhole_7129 := [[503.88, -35.49, 190.18], [0.217818, 0.672722, 0.696835, -0.120086], [0,0,0,0], [9E9, 9E9, 9E9, 9E9, 9E9, 9E9]];
	VAR robtarget Openhole_7130 := [[492.01, -36.34, 188.64], [0.190756, 0.680891, 0.702272, -0.082549], [0,0,0,0], [9E9, 9E9, 9E9, 9E9, 9E9, 9E9]];
	VAR robtarget Openhole_7131 := [[483.63, -37.25, 187.55], [0.170711, 0.686191, 0.705092, -0.053343], [0,0,0,0], [9E9, 9E9, 9E9, 9E9, 9E9, 9E9]];
	VAR robtarget Openhole_7132 := [[476.28, -38.4, 186.56], [0.153044, 0.690346, 0.706642, -0.025623], [0,0,0,0], [9E9, 9E9, 9E9, 9E9, 9E9, 9E9]];
	VAR robtarget Openhole_7133 := [[475.31, -38.59, 186.43], [0.15072, 0.690857, 0.706771, -0.021791], [0,0,0,0], [9E9, 9E9, 9E9, 9E9, 9E9, 9E9]];
	VAR robtarget Openhole_7134 := [[474.82, -38.7, 186.36], [0.149483, 0.691126, 0.706825, -0.019948], [0,0,0,0], [9E9, 9E9, 9E9, 9E9, 9E9, 9E9]];
	VAR robtarget Openhole_7135 := [[470.42, -38.7, 185.53], [0.136106, 0.693884, 0.707088, -0.005131], [0,0,0,0], [9E9, 9E9, 9E9, 9E9, 9E9, 9E9]];
	VAR robtarget Openhole_7136 := [[470.91, -38.55, 185.59], [0.137254, 0.693658, 0.707071, -0.007111], [0,0,0,0], [9E9, 9E9, 9E9, 9E9, 9E9, 9E9]];
	VAR robtarget Openhole_7137 := [[477.71, -37.2, 186.5], [0.153532, 0.690238, 0.70628, -0.034191], [0,0,0,0], [9E9, 9E9, 9E9, 9E9, 9E9, 9E9]];
	VAR robtarget Openhole_7138 := [[485.08, -36.14, 187.42], [0.171412, 0.686016, 0.704431, -0.061462], [0,0,0,0], [9E9, 9E9, 9E9, 9E9, 9E9, 9E9]];
	VAR robtarget Openhole_7139 := [[493.97, -35.28, 188.52], [0.192767, 0.680324, 0.70113, -0.091745], [0,0,0,0], [9E9, 9E9, 9E9, 9E9, 9E9, 9E9]];
	VAR robtarget Openhole_7140 := [[504.37, -34.58, 189.77], [0.216412, 0.673176, 0.696125, -0.124138], [0,0,0,0], [9E9, 9E9, 9E9, 9E9, 9E9, 9E9]];
	VAR robtarget Openhole_7141 := [[509.38, -34.58, 190.52], [0.183051, 0.683002, 0.683002, -0.183051], [0,0,0,0], [9E9, 9E9, 9E9, 9E9, 9E9, 9E9]];
	VAR robtarget Openhole_7142 := [[536.38, -34.58, 190.44], [0.183051, 0.683002, 0.683002, -0.183051], [0,0,0,0], [9E9, 9E9, 9E9, 9E9, 9E9, 9E9]];
	VAR robtarget Openhole_7143 := [[536.37, -33.69, 189.93], [0.183051, 0.683002, 0.683002, -0.183051], [0,0,0,0], [9E9, 9E9, 9E9, 9E9, 9E9, 9E9]];
	VAR robtarget Openhole_7144 := [[524.37, -33.69, 189.96], [0.183051, 0.683002, 0.683002, -0.183051], [0,0,0,0], [9E9, 9E9, 9E9, 9E9, 9E9, 9E9]];
	VAR robtarget Openhole_7145 := [[509.37, -33.69, 190.01], [0.183051, 0.683002, 0.683002, -0.183051], [0,0,0,0], [9E9, 9E9, 9E9, 9E9, 9E9, 9E9]];
	VAR robtarget Openhole_7146 := [[504.38, -33.69, 189.31], [0.213931, 0.673968, 0.69566, -0.126715], [0,0,0,0], [9E9, 9E9, 9E9, 9E9, 9E9, 9E9]];
	VAR robtarget Openhole_7147 := [[490, -34.71, 187.68], [0.18059, 0.683657, 0.702414, -0.081334], [0,0,0,0], [9E9, 9E9, 9E9, 9E9, 9E9, 9E9]];
	VAR robtarget Openhole_7148 := [[482.1, -35.58, 186.76], [0.161258, 0.688474, 0.705068, -0.053655], [0,0,0,0], [9E9, 9E9, 9E9, 9E9, 9E9, 9E9]];
	VAR robtarget Openhole_7149 := [[475.24, -36.68, 185.94], [0.144521, 0.69218, 0.706566, -0.02764], [0,0,0,0], [9E9, 9E9, 9E9, 9E9, 9E9, 9E9]];
	VAR robtarget Openhole_7150 := [[467.97, -38.24, 184.98], [0.127119, 0.695587, 0.707104, 0.001859], [0,0,0,0], [9E9, 9E9, 9E9, 9E9, 9E9, 9E9]];
	VAR robtarget Openhole_7151 := [[467, -38.47, 184.84], [0.124817, 0.696003, 0.707082, 0.005874], [0,0,0,0], [9E9, 9E9, 9E9, 9E9, 9E9, 9E9]];
	VAR robtarget Openhole_7152 := [[466.52, -38.7, 184.79], [0.123907, 0.696166, 0.70706, 0.008148], [0,0,0,0], [9E9, 9E9, 9E9, 9E9, 9E9, 9E9]];
	VAR robtarget Openhole_7153 := [[462.13, -38.7, 183.96], [0.109894, 0.698515, 0.706728, 0.02313], [0,0,0,0], [9E9, 9E9, 9E9, 9E9, 9E9, 9E9]];
	VAR robtarget Openhole_7154 := [[462.62, -38.48, 184.02], [0.110823, 0.698368, 0.706799, 0.020848], [0,0,0,0], [9E9, 9E9, 9E9, 9E9, 9E9, 9E9]];
	VAR robtarget Openhole_7155 := [[471.3, -36.44, 185.22], [0.131764, 0.694722, 0.706943, -0.015235], [0,0,0,0], [9E9, 9E9, 9E9, 9E9, 9E9, 9E9]];
	VAR robtarget Openhole_7156 := [[478.14, -35.16, 186.01], [0.148422, 0.691354, 0.705855, -0.042058], [0,0,0,0], [9E9, 9E9, 9E9, 9E9, 9E9, 9E9]];
	VAR robtarget Openhole_7157 := [[485.53, -34.21, 186.83], [0.166787, 0.687155, 0.703741, -0.068907], [0,0,0,0], [9E9, 9E9, 9E9, 9E9, 9E9, 9E9]];
	VAR robtarget Openhole_7158 := [[495.44, -33.39, 187.91], [0.190982, 0.680827, 0.699732, -0.101858], [0,0,0,0], [9E9, 9E9, 9E9, 9E9, 9E9, 9E9]];
	VAR robtarget Openhole_7159 := [[504.38, -32.81, 188.84], [0.211438, 0.674755, 0.695187, -0.129289], [0,0,0,0], [9E9, 9E9, 9E9, 9E9, 9E9, 9E9]];
	VAR robtarget Openhole_7160 := [[509.37, -32.81, 189.5], [0.183051, 0.683002, 0.683002, -0.183051], [0,0,0,0], [9E9, 9E9, 9E9, 9E9, 9E9, 9E9]];
	VAR robtarget Openhole_7161 := [[536.37, -32.81, 189.42], [0.183051, 0.683002, 0.683002, -0.183051], [0,0,0,0], [9E9, 9E9, 9E9, 9E9, 9E9, 9E9]];
	VAR robtarget Openhole_7162 := [[536.37, -31.93, 188.91], [0.183051, 0.683002, 0.683002, -0.183051], [0,0,0,0], [9E9, 9E9, 9E9, 9E9, 9E9, 9E9]];
	VAR robtarget Openhole_7163 := [[524.37, -31.93, 188.94], [0.183051, 0.683002, 0.683002, -0.183051], [0,0,0,0], [9E9, 9E9, 9E9, 9E9, 9E9, 9E9]];
	VAR robtarget Openhole_7164 := [[509.37, -31.93, 188.99], [0.183051, 0.683002, 0.683002, -0.183051], [0,0,0,0], [9E9, 9E9, 9E9, 9E9, 9E9, 9E9]];
	VAR robtarget Openhole_7165 := [[504.38, -31.93, 188.37], [0.208936, 0.675534, 0.694702, -0.131865], [0,0,0,0], [9E9, 9E9, 9E9, 9E9, 9E9, 9E9]];
	VAR robtarget Openhole_7166 := [[487.99, -33.03, 186.75], [0.170012, 0.686364, 0.702533, -0.080297], [0,0,0,0], [9E9, 9E9, 9E9, 9E9, 9E9, 9E9]];
	VAR robtarget Openhole_7167 := [[479.58, -33.93, 185.88], [0.148799, 0.691273, 0.705285, -0.05072], [0,0,0,0], [9E9, 9E9, 9E9, 9E9, 9E9, 9E9]];
	VAR robtarget Openhole_7168 := [[473.2, -34.93, 185.19], [0.132793, 0.694526, 0.706612, -0.026453], [0,0,0,0], [9E9, 9E9, 9E9, 9E9, 9E9, 9E9]];
	VAR robtarget Openhole_7169 := [[466.4, -36.39, 184.39], [0.116235, 0.697488, 0.707106, 0.00119], [0,0,0,0], [9E9, 9E9, 9E9, 9E9, 9E9, 9E9]];
	VAR robtarget Openhole_7170 := [[457.76, -38.56, 183.12], [0.095196, 0.700669, 0.706099, 0.037734], [0,0,0,0], [9E9, 9E9, 9E9, 9E9, 9E9, 9E9]];
	VAR robtarget Openhole_7171 := [[457.28, -38.7, 183.04], [0.094014, 0.700829, 0.705988, 0.039769], [0,0,0,0], [9E9, 9E9, 9E9, 9E9, 9E9, 9E9]];
	VAR robtarget Openhole_7172 := [[452.92, -38.7, 182.22], [0.079521, 0.702621, 0.704992, 0.054647], [0,0,0,0], [9E9, 9E9, 9E9, 9E9, 9E9, 9E9]];
	VAR robtarget Openhole_7173 := [[460.54, -36.57, 183.43], [0.097896, 0.700297, 0.706773, 0.021731], [0,0,0,0], [9E9, 9E9, 9E9, 9E9, 9E9, 9E9]];
	VAR robtarget Openhole_7174 := [[467.77, -34.81, 184.34], [0.115488, 0.697612, 0.707054, -0.008633], [0,0,0,0], [9E9, 9E9, 9E9, 9E9, 9E9, 9E9]];
	VAR robtarget Openhole_7175 := [[474.13, -33.64, 185.03], [0.131523, 0.694767, 0.706302, -0.033737], [0,0,0,0], [9E9, 9E9, 9E9, 9E9, 9E9, 9E9]];
	VAR robtarget Openhole_7176 := [[481.53, -32.67, 185.76], [0.150556, 0.690893, 0.704469, -0.061024], [0,0,0,0], [9E9, 9E9, 9E9, 9E9, 9E9, 9E9]];
	VAR robtarget Openhole_7177 := [[491.44, -31.83, 186.73], [0.175806, 0.684903, 0.700746, -0.094632], [0,0,0,0], [9E9, 9E9, 9E9, 9E9, 9E9, 9E9]];
	VAR robtarget Openhole_7178 := [[504.38, -31.04, 187.9], [0.206434, 0.676302, 0.694207, -0.134452], [0,0,0,0], [9E9, 9E9, 9E9, 9E9, 9E9, 9E9]];
	VAR robtarget Openhole_7179 := [[509.37, -31.04, 188.48], [0.183051, 0.683002, 0.683002, -0.183051], [0,0,0,0], [9E9, 9E9, 9E9, 9E9, 9E9, 9E9]];
	VAR robtarget Openhole_7180 := [[536.33, -31.04, 188.4], [0.183051, 0.683002, 0.683002, -0.183051], [0,0,0,0], [9E9, 9E9, 9E9, 9E9, 9E9, 9E9]];
	VAR robtarget Openhole_7181 := [[536.24, -21.49, 182.88], [0.183051, 0.683002, 0.683002, -0.183051], [0,0,0,0], [9E9, 9E9, 9E9, 9E9, 9E9, 9E9]];
	VAR robtarget Openhole_7182 := [[509.35, -21.49, 182.97], [0.183051, 0.683002, 0.683002, -0.183051], [0,0,0,0], [9E9, 9E9, 9E9, 9E9, 9E9, 9E9]];
	VAR robtarget Openhole_7183 := [[504.35, -21.49, 182.85], [0.178856, 0.684113, 0.688234, -0.162275], [0,0,0,0], [9E9, 9E9, 9E9, 9E9, 9E9, 9E9]];
	VAR robtarget Openhole_7184 := [[503.38, -21.52, 182.84], [0.176485, 0.684728, 0.688851, -0.159636], [0,0,0,0], [9E9, 9E9, 9E9, 9E9, 9E9, 9E9]];
	VAR robtarget Openhole_7185 := [[493.89, -21.85, 182.75], [0.15215, 0.690544, 0.694572, -0.132552], [0,0,0,0], [9E9, 9E9, 9E9, 9E9, 9E9, 9E9]];
	VAR robtarget Openhole_7186 := [[487.39, -21.9, 182.59], [0.133831, 0.694326, 0.697957, -0.113387], [0,0,0,0], [9E9, 9E9, 9E9, 9E9, 9E9, 9E9]];
	VAR robtarget Openhole_7187 := [[486.89, -21.89, 182.58], [0.13237, 0.694606, 0.698198, -0.111891], [0,0,0,0], [9E9, 9E9, 9E9, 9E9, 9E9, 9E9]];
	VAR robtarget Openhole_7188 := [[473.4, -21.68, 182.16], [0.090397, 0.701305, 0.703588, -0.070458], [0,0,0,0], [9E9, 9E9, 9E9, 9E9, 9E9, 9E9]];
	VAR robtarget Openhole_7189 := [[465.92, -21.31, 181.91], [0.0649, 0.704122, 0.705533, -0.047149], [0,0,0,0], [9E9, 9E9, 9E9, 9E9, 9E9, 9E9]];
	VAR robtarget Openhole_7190 := [[463.93, -21.12, 181.84], [0.057682, 0.70475, 0.705908, -0.041162], [0,0,0,0], [9E9, 9E9, 9E9, 9E9, 9E9, 9E9]];
	VAR robtarget Openhole_7191 := [[457.02, -21.12, 181.7], [0.034525, 0.706263, 0.706879, -0.017953], [0,0,0,0], [9E9, 9E9, 9E9, 9E9, 9E9, 9E9]];
	VAR robtarget Openhole_7192 := [[456.81, -15.81, 181.31], [0.015738, 0.706932, 0.70623, -0.035197], [0,0,0,0], [9E9, 9E9, 9E9, 9E9, 9E9, 9E9]];
	VAR robtarget Openhole_7193 := [[457.68, -15.38, 181.25], [0.017254, 0.706896, 0.705997, -0.039604], [0,0,0,0], [9E9, 9E9, 9E9, 9E9, 9E9, 9E9]];
	VAR robtarget Openhole_7194 := [[458.51, -14.82, 181.17], [0.01814, 0.706874, 0.70572, -0.044262], [0,0,0,0], [9E9, 9E9, 9E9, 9E9, 9E9, 9E9]];
	VAR robtarget Openhole_7195 := [[460.62, -13.5, 180.94], [0.02086, 0.706799, 0.704906, -0.055743], [0,0,0,0], [9E9, 9E9, 9E9, 9E9, 9E9, 9E9]];
	VAR robtarget Openhole_7196 := [[461.06, -13.27, 180.89], [0.02157, 0.706778, 0.704725, -0.057984], [0,0,0,0], [9E9, 9E9, 9E9, 9E9, 9E9, 9E9]];
	VAR robtarget Openhole_7197 := [[460.89, -17, 181.32], [0.033598, 0.706308, 0.705681, -0.044878], [0,0,0,0], [9E9, 9E9, 9E9, 9E9, 9E9, 9E9]];
	VAR robtarget Openhole_7198 := [[462.52, -15.87, 181.14], [0.035264, 0.706227, 0.70503, -0.054149], [0,0,0,0], [9E9, 9E9, 9E9, 9E9, 9E9, 9E9]];
	VAR robtarget Openhole_7199 := [[462.94, -15.6, 181.09], [0.035767, 0.706202, 0.704851, -0.056441], [0,0,0,0], [9E9, 9E9, 9E9, 9E9, 9E9, 9E9]];
	VAR robtarget Openhole_7200 := [[463.8, -15.08, 180.99], [0.036891, 0.706144, 0.704472, -0.060983], [0,0,0,0], [9E9, 9E9, 9E9, 9E9, 9E9, 9E9]];
	VAR robtarget Openhole_7201 := [[464.66, -14.6, 180.89], [0.038172, 0.706076, 0.70407, -0.065467], [0,0,0,0], [9E9, 9E9, 9E9, 9E9, 9E9, 9E9]];
	VAR robtarget Openhole_7202 := [[465.55, -14.15, 180.78], [0.039638, 0.705995, 0.703646, -0.069876], [0,0,0,0], [9E9, 9E9, 9E9, 9E9, 9E9, 9E9]];
	VAR robtarget Openhole_7203 := [[466, -13.94, 180.73], [0.040444, 0.705949, 0.703427, -0.07205], [0,0,0,0], [9E9, 9E9, 9E9, 9E9, 9E9, 9E9]];
	VAR robtarget Openhole_7204 := [[466.46, -13.74, 180.67], [0.041292, 0.7059, 0.703203, -0.074201], [0,0,0,0], [9E9, 9E9, 9E9, 9E9, 9E9, 9E9]];
	VAR robtarget Openhole_7205 := [[467.38, -13.37, 180.56], [0.043131, 0.70579, 0.702743, -0.078433], [0,0,0,0], [9E9, 9E9, 9E9, 9E9, 9E9, 9E9]];
	VAR robtarget Openhole_7206 := [[467.85, -13.2, 180.5], [0.044111, 0.70573, 0.702508, -0.080515], [0,0,0,0], [9E9, 9E9, 9E9, 9E9, 9E9, 9E9]];
	VAR robtarget Openhole_7207 := [[468.32, -13.04, 180.45], [0.04515, 0.705664, 0.70227, -0.082563], [0,0,0,0], [9E9, 9E9, 9E9, 9E9, 9E9, 9E9]];
	VAR robtarget Openhole_7208 := [[469.27, -12.75, 180.34], [0.047333, 0.705521, 0.701785, -0.086591], [0,0,0,0], [9E9, 9E9, 9E9, 9E9, 9E9, 9E9]];
	VAR robtarget Openhole_7209 := [[470.71, -12.36, 180.17], [0.050807, 0.705279, 0.701033, -0.092482], [0,0,0,0], [9E9, 9E9, 9E9, 9E9, 9E9, 9E9]];
	VAR robtarget Openhole_7210 := [[471.19, -12.25, 180.12], [0.052033, 0.70519, 0.700778, -0.094393], [0,0,0,0], [9E9, 9E9, 9E9, 9E9, 9E9, 9E9]];
	VAR robtarget Openhole_7211 := [[471.68, -12.15, 180.06], [0.053298, 0.705095, 0.700522, -0.096275], [0,0,0,0], [9E9, 9E9, 9E9, 9E9, 9E9, 9E9]];
	VAR robtarget Openhole_7212 := [[475.61, -11.57, 179.66], [0.064235, 0.704183, 0.698415, -0.11053], [0,0,0,0], [9E9, 9E9, 9E9, 9E9, 9E9, 9E9]];
	VAR robtarget Openhole_7213 := [[480.09, -11.3, 179.26], [0.077724, 0.702822, 0.695957, -0.125075], [0,0,0,0], [9E9, 9E9, 9E9, 9E9, 9E9, 9E9]];
	VAR robtarget Openhole_7214 := [[482.58, -11.27, 179.06], [0.085491, 0.70192, 0.694558, -0.132622], [0,0,0,0], [9E9, 9E9, 9E9, 9E9, 9E9, 9E9]];
	VAR robtarget Openhole_7215 := [[483.08, -11.27, 179.02], [0.087054, 0.701728, 0.694276, -0.134095], [0,0,0,0], [9E9, 9E9, 9E9, 9E9, 9E9, 9E9]];
	VAR robtarget Openhole_7216 := [[497.54, -11.57, 178.08], [0.131094, 0.694848, 0.685443, -0.17369], [0,0,0,0], [9E9, 9E9, 9E9, 9E9, 9E9, 9E9]];
	VAR robtarget Openhole_7217 := [[498.04, -11.57, 178.04], [0.132496, 0.694583, 0.685107, -0.175009], [0,0,0,0], [9E9, 9E9, 9E9, 9E9, 9E9, 9E9]];
	VAR robtarget Openhole_7218 := [[503.02, -11.41, 177.6], [0.14577, 0.691919, 0.681584, -0.188263], [0,0,0,0], [9E9, 9E9, 9E9, 9E9, 9E9, 9E9]];
	VAR robtarget Openhole_7219 := [[503.51, -11.37, 177.55], [0.147018, 0.691654, 0.681215, -0.189596], [0,0,0,0], [9E9, 9E9, 9E9, 9E9, 9E9, 9E9]];
	VAR robtarget Openhole_7220 := [[504.33, -11.35, 177.48], [0.149152, 0.691197, 0.680624, -0.191706], [0,0,0,0], [9E9, 9E9, 9E9, 9E9, 9E9, 9E9]];
	VAR robtarget Openhole_7221 := [[509.33, -11.35, 177.11], [0.183051, 0.683002, 0.683002, -0.183051], [0,0,0,0], [9E9, 9E9, 9E9, 9E9, 9E9, 9E9]];
	VAR robtarget Openhole_7222 := [[536.33, -11.35, 177.02], [0.183051, 0.683002, 0.683002, -0.183051], [0,0,0,0], [9E9, 9E9, 9E9, 9E9, 9E9, 9E9]];
	VAR robtarget Openhole_7223 := [[536.34, -13.35, 178.18], [0.183051, 0.683002, 0.683002, -0.183051], [0,0,0,0], [9E9, 9E9, 9E9, 9E9, 9E9, 9E9]];
	VAR robtarget Openhole_7224 := [[509.34, -13.35, 178.26], [0.183051, 0.683002, 0.683002, -0.183051], [0,0,0,0], [9E9, 9E9, 9E9, 9E9, 9E9, 9E9]];
	VAR robtarget Openhole_7225 := [[504.34, -13.35, 178.53], [0.155015, 0.689906, 0.68222, -0.185947], [0,0,0,0], [9E9, 9E9, 9E9, 9E9, 9E9, 9E9]];
	VAR robtarget Openhole_7226 := [[498.25, -13.65, 179.01], [0.139367, 0.693237, 0.686525, -0.169362], [0,0,0,0], [9E9, 9E9, 9E9, 9E9, 9E9, 9E9]];
	VAR robtarget Openhole_7227 := [[494.76, -13.69, 179.21], [0.129618, 0.695125, 0.688803, -0.159846], [0,0,0,0], [9E9, 9E9, 9E9, 9E9, 9E9, 9E9]];
	VAR robtarget Openhole_7228 := [[494.26, -13.69, 179.23], [0.128186, 0.695391, 0.689118, -0.15848], [0,0,0,0], [9E9, 9E9, 9E9, 9E9, 9E9, 9E9]];
	VAR robtarget Openhole_7229 := [[482.27, -13.53, 179.8], [0.091773, 0.701126, 0.69605, -0.124555], [0,0,0,0], [9E9, 9E9, 9E9, 9E9, 9E9, 9E9]];
	VAR robtarget Openhole_7230 := [[481.77, -13.53, 179.83], [0.090218, 0.701328, 0.696317, -0.123054], [0,0,0,0], [9E9, 9E9, 9E9, 9E9, 9E9, 9E9]];
	VAR robtarget Openhole_7231 := [[476.29, -13.68, 180.15], [0.073319, 0.703295, 0.69915, -0.105779], [0,0,0,0], [9E9, 9E9, 9E9, 9E9, 9E9, 9E9]];
	VAR robtarget Openhole_7232 := [[474.3, -13.82, 180.29], [0.06737, 0.70389, 0.700131, -0.099082], [0,0,0,0], [9E9, 9E9, 9E9, 9E9, 9E9, 9E9]];
	VAR robtarget Openhole_7233 := [[473.3, -13.93, 180.37], [0.064515, 0.704158, 0.700615, -0.095593], [0,0,0,0], [9E9, 9E9, 9E9, 9E9, 9E9, 9E9]];
	VAR robtarget Openhole_7234 := [[470.86, -19.93, 181.73], [0.076428, 0.702964, 0.70383, -0.067992], [0,0,0,0], [9E9, 9E9, 9E9, 9E9, 9E9, 9E9]];
	VAR robtarget Openhole_7235 := [[487.35, -20.27, 181.99], [0.128586, 0.695317, 0.697126, -0.118388], [0,0,0,0], [9E9, 9E9, 9E9, 9E9, 9E9, 9E9]];
	VAR robtarget Openhole_7236 := [[489.35, -20.27, 182.02], [0.13443, 0.694211, 0.6961, -0.124277], [0,0,0,0], [9E9, 9E9, 9E9, 9E9, 9E9, 9E9]];
	VAR robtarget Openhole_7237 := [[489.85, -20.27, 182.03], [0.135872, 0.69393, 0.695837, -0.125742], [0,0,0,0], [9E9, 9E9, 9E9, 9E9, 9E9, 9E9]];
	VAR robtarget Openhole_7238 := [[499.85, -20.1, 182.06], [0.163043, 0.688053, 0.690041, -0.154414], [0,0,0,0], [9E9, 9E9, 9E9, 9E9, 9E9, 9E9]];
	VAR robtarget Openhole_7239 := [[504.35, -19.88, 182], [0.174161, 0.685323, 0.687111, -0.16697], [0,0,0,0], [9E9, 9E9, 9E9, 9E9, 9E9, 9E9]];
	VAR robtarget Openhole_7240 := [[536.35, -19.88, 181.95], [0.183051, 0.683002, 0.683002, -0.183051], [0,0,0,0], [9E9, 9E9, 9E9, 9E9, 9E9, 9E9]];
	VAR robtarget Openhole_7241 := [[536.35, -19.19, 181.55], [0.183051, 0.683002, 0.683002, -0.183051], [0,0,0,0], [9E9, 9E9, 9E9, 9E9, 9E9, 9E9]];
	VAR robtarget Openhole_7242 := [[509.35, -19.19, 181.63], [0.183051, 0.683002, 0.683002, -0.183051], [0,0,0,0], [9E9, 9E9, 9E9, 9E9, 9E9, 9E9]];
	VAR robtarget Openhole_7243 := [[504.35, -19.19, 181.63], [0.172124, 0.685838, 0.686614, -0.169002], [0,0,0,0], [9E9, 9E9, 9E9, 9E9, 9E9, 9E9]];
	VAR robtarget Openhole_7244 := [[495.63, -19.51, 181.76], [0.149838, 0.691049, 0.692163, -0.144602], [0,0,0,0], [9E9, 9E9, 9E9, 9E9, 9E9, 9E9]];
	VAR robtarget Openhole_7245 := [[490.13, -19.56, 181.75], [0.134457, 0.694206, 0.695281, -0.128783], [0,0,0,0], [9E9, 9E9, 9E9, 9E9, 9E9, 9E9]];
	VAR robtarget Openhole_7246 := [[489.63, -19.56, 181.75], [0.13301, 0.694484, 0.695548, -0.127328], [0,0,0,0], [9E9, 9E9, 9E9, 9E9, 9E9, 9E9]];
	VAR robtarget Openhole_7247 := [[470.13, -19.24, 181.58], [0.071794, 0.703453, 0.703837, -0.067927], [0,0,0,0], [9E9, 9E9, 9E9, 9E9, 9E9, 9E9]];
	VAR robtarget Openhole_7248 := [[469.63, -19.24, 181.58], [0.070166, 0.703617, 0.703992, -0.066296], [0,0,0,0], [9E9, 9E9, 9E9, 9E9, 9E9, 9E9]];
	VAR robtarget Openhole_7249 := [[469.13, -19.24, 181.58], [0.068526, 0.703779, 0.704143, -0.064671], [0,0,0,0], [9E9, 9E9, 9E9, 9E9, 9E9, 9E9]];
	VAR robtarget Openhole_7250 := [[466.64, -19.31, 181.59], [0.060557, 0.704509, 0.704868, -0.056227], [0,0,0,0], [9E9, 9E9, 9E9, 9E9, 9E9, 9E9]];
	VAR robtarget Openhole_7251 := [[466.14, -19.31, 181.59], [0.058918, 0.704648, 0.704998, -0.054563], [0,0,0,0], [9E9, 9E9, 9E9, 9E9, 9E9, 9E9]];
	VAR robtarget Openhole_7252 := [[465.64, -19.33, 181.59], [0.057316, 0.70478, 0.705128, -0.05286], [0,0,0,0], [9E9, 9E9, 9E9, 9E9, 9E9, 9E9]];
	VAR robtarget Openhole_7253 := [[464.64, -19.38, 181.59], [0.054189, 0.705027, 0.705381, -0.049366], [0,0,0,0], [9E9, 9E9, 9E9, 9E9, 9E9, 9E9]];
	VAR robtarget Openhole_7254 := [[464.14, -19.42, 181.6], [0.052664, 0.705143, 0.705504, -0.047577], [0,0,0,0], [9E9, 9E9, 9E9, 9E9, 9E9, 9E9]];
	VAR robtarget Openhole_7255 := [[463.64, -19.43, 181.6], [0.051023, 0.705264, 0.705616, -0.04589], [0,0,0,0], [9E9, 9E9, 9E9, 9E9, 9E9, 9E9]];
	VAR robtarget Openhole_7256 := [[462.64, -19.54, 181.61], [0.048059, 0.705472, 0.705845, -0.042221], [0,0,0,0], [9E9, 9E9, 9E9, 9E9, 9E9, 9E9]];
	VAR robtarget Openhole_7257 := [[462.15, -19.58, 181.61], [0.046533, 0.705574, 0.705951, -0.040416], [0,0,0,0], [9E9, 9E9, 9E9, 9E9, 9E9, 9E9]];
	VAR robtarget Openhole_7258 := [[461.97, -18.21, 181.44], [0.041318, 0.705899, 0.705709, -0.044435], [0,0,0,0], [9E9, 9E9, 9E9, 9E9, 9E9, 9E9]];
	VAR robtarget Openhole_7259 := [[462.42, -18, 181.41], [0.042124, 0.705851, 0.705566, -0.046651], [0,0,0,0], [9E9, 9E9, 9E9, 9E9, 9E9, 9E9]];
	VAR robtarget Openhole_7260 := [[462.86, -17.76, 181.38], [0.042807, 0.70581, 0.705414, -0.048906], [0,0,0,0], [9E9, 9E9, 9E9, 9E9, 9E9, 9E9]];
	VAR robtarget Openhole_7261 := [[463.78, -17.37, 181.31], [0.044575, 0.7057, 0.705098, -0.053262], [0,0,0,0], [9E9, 9E9, 9E9, 9E9, 9E9, 9E9]];
	VAR robtarget Openhole_7262 := [[465.15, -16.77, 181.2], [0.047091, 0.705537, 0.704572, -0.059818], [0,0,0,0], [9E9, 9E9, 9E9, 9E9, 9E9, 9E9]];
	VAR robtarget Openhole_7263 := [[465.61, -16.58, 181.16], [0.047984, 0.705477, 0.704386, -0.061973], [0,0,0,0], [9E9, 9E9, 9E9, 9E9, 9E9, 9E9]];
	VAR robtarget Openhole_7264 := [[466.54, -16.21, 181.08], [0.049857, 0.705347, 0.703998, -0.066232], [0,0,0,0], [9E9, 9E9, 9E9, 9E9, 9E9, 9E9]];
	VAR robtarget Openhole_7265 := [[467.01, -16.05, 181.04], [0.050861, 0.705275, 0.703798, -0.068324], [0,0,0,0], [9E9, 9E9, 9E9, 9E9, 9E9, 9E9]];
	VAR robtarget Openhole_7266 := [[468.44, -15.62, 180.92], [0.054179, 0.705028, 0.70318, -0.074416], [0,0,0,0], [9E9, 9E9, 9E9, 9E9, 9E9, 9E9]];
	VAR robtarget Openhole_7267 := [[469.41, -15.37, 180.84], [0.056526, 0.704844, 0.70275, -0.078376], [0,0,0,0], [9E9, 9E9, 9E9, 9E9, 9E9, 9E9]];
	VAR robtarget Openhole_7268 := [[471.36, -14.97, 180.68], [0.06161, 0.704418, 0.701859, -0.085987], [0,0,0,0], [9E9, 9E9, 9E9, 9E9, 9E9, 9E9]];
	VAR robtarget Openhole_7269 := [[471.85, -14.89, 180.65], [0.062952, 0.704299, 0.701631, -0.087828], [0,0,0,0], [9E9, 9E9, 9E9, 9E9, 9E9, 9E9]];
	VAR robtarget Openhole_7270 := [[472.35, -14.82, 180.61], [0.06433, 0.704174, 0.701402, -0.089636], [0,0,0,0], [9E9, 9E9, 9E9, 9E9, 9E9, 9E9]];
	VAR robtarget Openhole_7271 := [[476.32, -14.47, 180.36], [0.076031, 0.703007, 0.699518, -0.103318], [0,0,0,0], [9E9, 9E9, 9E9, 9E9, 9E9, 9E9]];
	VAR robtarget Openhole_7272 := [[480.81, -14.37, 180.13], [0.089945, 0.701363, 0.697282, -0.117462], [0,0,0,0], [9E9, 9E9, 9E9, 9E9, 9E9, 9E9]];
	VAR robtarget Openhole_7273 := [[481.31, -14.37, 180.11], [0.091508, 0.701161, 0.697026, -0.118973], [0,0,0,0], [9E9, 9E9, 9E9, 9E9, 9E9, 9E9]];
	VAR robtarget Openhole_7274 := [[493.8, -14.52, 179.61], [0.129424, 0.695161, 0.689974, -0.154712], [0,0,0,0], [9E9, 9E9, 9E9, 9E9, 9E9, 9E9]];
	VAR robtarget Openhole_7275 := [[494.3, -14.52, 179.59], [0.130854, 0.694894, 0.689664, -0.15609], [0,0,0,0], [9E9, 9E9, 9E9, 9E9, 9E9, 9E9]];
	VAR robtarget Openhole_7276 := [[501.29, -14.35, 179.2], [0.149795, 0.691058, 0.685043, -0.175259], [0,0,0,0], [9E9, 9E9, 9E9, 9E9, 9E9, 9E9]];
	VAR robtarget Openhole_7277 := [[504.34, -14.15, 178.96], [0.157364, 0.689374, 0.682846, -0.183634], [0,0,0,0], [9E9, 9E9, 9E9, 9E9, 9E9, 9E9]];
	VAR robtarget Openhole_7278 := [[509.34, -14.15, 178.72], [0.183051, 0.683002, 0.683002, -0.183051], [0,0,0,0], [9E9, 9E9, 9E9, 9E9, 9E9, 9E9]];
	VAR robtarget Openhole_7279 := [[536.34, -14.15, 178.64], [0.183051, 0.683002, 0.683002, -0.183051], [0,0,0,0], [9E9, 9E9, 9E9, 9E9, 9E9, 9E9]];
	VAR robtarget Openhole_7280 := [[536.34, -15.36, 179.34], [0.183051, 0.683002, 0.683002, -0.183051], [0,0,0,0], [9E9, 9E9, 9E9, 9E9, 9E9, 9E9]];
	VAR robtarget Openhole_7281 := [[509.34, -15.36, 179.42], [0.183051, 0.683002, 0.683002, -0.183051], [0,0,0,0], [9E9, 9E9, 9E9, 9E9, 9E9, 9E9]];
	VAR robtarget Openhole_7282 := [[504.34, -15.36, 179.6], [0.160909, 0.688555, 0.683778, -0.180133], [0,0,0,0], [9E9, 9E9, 9E9, 9E9, 9E9, 9E9]];
	VAR robtarget Openhole_7283 := [[503.64, -15.39, 179.64], [0.159169, 0.68896, 0.684266, -0.178269], [0,0,0,0], [9E9, 9E9, 9E9, 9E9, 9E9, 9E9]];
	VAR robtarget Openhole_7284 := [[497.66, -15.67, 179.98], [0.143827, 0.692325, 0.688358, -0.161751], [0,0,0,0], [9E9, 9E9, 9E9, 9E9, 9E9, 9E9]];
	VAR robtarget Openhole_7285 := [[492.67, -15.73, 180.17], [0.129897, 0.695073, 0.69148, -0.147838], [0,0,0,0], [9E9, 9E9, 9E9, 9E9, 9E9, 9E9]];
	VAR robtarget Openhole_7286 := [[492.17, -15.73, 180.18], [0.128453, 0.695342, 0.691778, -0.146436], [0,0,0,0], [9E9, 9E9, 9E9, 9E9, 9E9, 9E9]];
	VAR robtarget Openhole_7287 := [[479.17, -15.58, 180.55], [0.088709, 0.70152, 0.698724, -0.108559], [0,0,0,0], [9E9, 9E9, 9E9, 9E9, 9E9, 9E9]];
	VAR robtarget Openhole_7288 := [[478.67, -15.58, 180.57], [0.087137, 0.701717, 0.698962, -0.107015], [0,0,0,0], [9E9, 9E9, 9E9, 9E9, 9E9, 9E9]];
	VAR robtarget Openhole_7289 := [[473.18, -15.79, 180.8], [0.070251, 0.703608, 0.701468, -0.089122], [0,0,0,0], [9E9, 9E9, 9E9, 9E9, 9E9, 9E9]];
	VAR robtarget Openhole_7290 := [[472.19, -15.88, 180.85], [0.067309, 0.703896, 0.701899, -0.085659], [0,0,0,0], [9E9, 9E9, 9E9, 9E9, 9E9, 9E9]];
	VAR robtarget Openhole_7291 := [[470.21, -16.14, 180.96], [0.061706, 0.704409, 0.702743, -0.078438], [0,0,0,0], [9E9, 9E9, 9E9, 9E9, 9E9, 9E9]];
	VAR robtarget Openhole_7292 := [[469.72, -16.22, 180.99], [0.060381, 0.704524, 0.70295, -0.076562], [0,0,0,0], [9E9, 9E9, 9E9, 9E9, 9E9, 9E9]];
	VAR robtarget Openhole_7293 := [[469.23, -16.32, 181.02], [0.059092, 0.704633, 0.703155, -0.074656], [0,0,0,0], [9E9, 9E9, 9E9, 9E9, 9E9, 9E9]];
	VAR robtarget Openhole_7294 := [[468.25, -16.53, 181.09], [0.05659, 0.704839, 0.703556, -0.070778], [0,0,0,0], [9E9, 9E9, 9E9, 9E9, 9E9, 9E9]];
	VAR robtarget Openhole_7295 := [[467.28, -16.77, 181.15], [0.054178, 0.705028, 0.703942, -0.066824], [0,0,0,0], [9E9, 9E9, 9E9, 9E9, 9E9, 9E9]];
	VAR robtarget Openhole_7296 := [[466.6, -18.47, 181.45], [0.057641, 0.704754, 0.704649, -0.058904], [0,0,0,0], [9E9, 9E9, 9E9, 9E9, 9E9, 9E9]];
	VAR robtarget Openhole_7297 := [[467.1, -18.42, 181.44], [0.059091, 0.704633, 0.704494, -0.060728], [0,0,0,0], [9E9, 9E9, 9E9, 9E9, 9E9, 9E9]];
	VAR robtarget Openhole_7298 := [[469.59, -18.24, 181.39], [0.066681, 0.703956, 0.703685, -0.069483], [0,0,0,0], [9E9, 9E9, 9E9, 9E9, 9E9, 9E9]];
	VAR robtarget Openhole_7299 := [[471.09, -18.16, 181.36], [0.071308, 0.703502, 0.703161, -0.074598], [0,0,0,0], [9E9, 9E9, 9E9, 9E9, 9E9, 9E9]];
	VAR robtarget Openhole_7300 := [[474.59, -18.11, 181.32], [0.082432, 0.702286, 0.701859, -0.085985], [0,0,0,0], [9E9, 9E9, 9E9, 9E9, 9E9, 9E9]];
	VAR robtarget Openhole_7301 := [[475.09, -18.11, 181.31], [0.084036, 0.702095, 0.701664, -0.087566], [0,0,0,0], [9E9, 9E9, 9E9, 9E9, 9E9, 9E9]];
	VAR robtarget Openhole_7302 := [[491.09, -18.34, 181.27], [0.133427, 0.694404, 0.694038, -0.135319], [0,0,0,0], [9E9, 9E9, 9E9, 9E9, 9E9, 9E9]];
	VAR robtarget Openhole_7303 := [[491.59, -18.34, 181.26], [0.134863, 0.694127, 0.693757, -0.136752], [0,0,0,0], [9E9, 9E9, 9E9, 9E9, 9E9, 9E9]];
	VAR robtarget Openhole_7304 := [[500.08, -18.17, 181.12], [0.157931, 0.689244, 0.688586, -0.160778], [0,0,0,0], [9E9, 9E9, 9E9, 9E9, 9E9, 9E9]];
	VAR robtarget Openhole_7305 := [[504.35, -17.96, 180.98], [0.168544, 0.686726, 0.685727, -0.172565], [0,0,0,0], [9E9, 9E9, 9E9, 9E9, 9E9, 9E9]];
	VAR robtarget Openhole_7306 := [[536.35, -17.96, 180.84], [0.183051, 0.683002, 0.683002, -0.183051], [0,0,0,0], [9E9, 9E9, 9E9, 9E9, 9E9, 9E9]];
	VAR robtarget Openhole_7307 := [[536.34, -17.24, 180.42], [0.183051, 0.683002, 0.683002, -0.183051], [0,0,0,0], [9E9, 9E9, 9E9, 9E9, 9E9, 9E9]];
	VAR robtarget Openhole_7308 := [[509.34, -17.24, 180.51], [0.183051, 0.683002, 0.683002, -0.183051], [0,0,0,0], [9E9, 9E9, 9E9, 9E9, 9E9, 9E9]];
	VAR robtarget Openhole_7309 := [[504.34, -17.24, 180.6], [0.16643, 0.687242, 0.685195, -0.174664], [0,0,0,0], [9E9, 9E9, 9E9, 9E9, 9E9, 9E9]];
	VAR robtarget Openhole_7310 := [[503.53, -17.27, 180.63], [0.164404, 0.687729, 0.685747, -0.172486], [0,0,0,0], [9E9, 9E9, 9E9, 9E9, 9E9, 9E9]];
	VAR robtarget Openhole_7311 := [[496.04, -17.57, 180.89], [0.145093, 0.692061, 0.69066, -0.151622], [0,0,0,0], [9E9, 9E9, 9E9, 9E9, 9E9, 9E9]];
	VAR robtarget Openhole_7312 := [[491.04, -17.63, 180.98], [0.13109, 0.694849, 0.693627, -0.137409], [0,0,0,0], [9E9, 9E9, 9E9, 9E9, 9E9, 9E9]];
	VAR robtarget Openhole_7313 := [[490.54, -17.62, 180.99], [0.129642, 0.695121, 0.69391, -0.135975], [0,0,0,0], [9E9, 9E9, 9E9, 9E9, 9E9, 9E9]];
	VAR robtarget Openhole_7314 := [[481.55, -17.51, 181.07], [0.102326, 0.699664, 0.698553, -0.109655], [0,0,0,0], [9E9, 9E9, 9E9, 9E9, 9E9, 9E9]];
	VAR robtarget Openhole_7315 := [[483.56, -27.51, 184.34], [0.14032, 0.693044, 0.702115, -0.083872], [0,0,0,0], [9E9, 9E9, 9E9, 9E9, 9E9, 9E9]];
	VAR robtarget Openhole_7316 := [[469.62, -28.25, 183.34], [0.099934, 0.700009, 0.706169, -0.036396], [0,0,0,0], [9E9, 9E9, 9E9, 9E9, 9E9, 9E9]];
	VAR robtarget Openhole_7317 := [[459.18, -29.01, 182.49], [0.068385, 0.703792, 0.707106, 0.00128], [0,0,0,0], [9E9, 9E9, 9E9, 9E9, 9E9, 9E9]];
	VAR robtarget Openhole_7318 := [[458.68, -29.06, 182.44], [0.066901, 0.703935, 0.7071, 0.003132], [0,0,0,0], [9E9, 9E9, 9E9, 9E9, 9E9, 9E9]];
	VAR robtarget Openhole_7319 := [[453.24, -29.67, 181.94], [0.05065, 0.70529, 0.70671, 0.023675], [0,0,0,0], [9E9, 9E9, 9E9, 9E9, 9E9, 9E9]];
	VAR robtarget Openhole_7320 := [[451.75, -29.75, 181.79], [0.045868, 0.705618, 0.706512, 0.029007], [0,0,0,0], [9E9, 9E9, 9E9, 9E9, 9E9, 9E9]];
	VAR robtarget Openhole_7321 := [[451.25, -29.75, 181.74], [0.04419, 0.705725, 0.70644, 0.030706], [0,0,0,0], [9E9, 9E9, 9E9, 9E9, 9E9, 9E9]];
	VAR robtarget Openhole_7322 := [[450.76, -29.75, 181.69], [0.042497, 0.705829, 0.706364, 0.032391], [0,0,0,0], [9E9, 9E9, 9E9, 9E9, 9E9, 9E9]];
	VAR robtarget Openhole_7323 := [[443.3, -29.47, 180.93], [0.016101, 0.706923, 0.704837, 0.056611], [0,0,0,0], [9E9, 9E9, 9E9, 9E9, 9E9, 9E9]];
	VAR robtarget Openhole_7324 := [[441.81, -29.49, 180.78], [0.011075, 0.70702, 0.704412, 0.061674], [0,0,0,0], [9E9, 9E9, 9E9, 9E9, 9E9, 9E9]];
	VAR robtarget Openhole_7325 := [[439.82, -29.61, 180.57], [0.004681, 0.707091, 0.703765, 0.068668], [0,0,0,0], [9E9, 9E9, 9E9, 9E9, 9E9, 9E9]];
	VAR robtarget Openhole_7326 := [[437.85, -29.84, 180.35], [-0.001272, 0.707106, 0.703015, 0.075964], [0,0,0,0], [9E9, 9E9, 9E9, 9E9, 9E9, 9E9]];
	VAR robtarget Openhole_7327 := [[428.05, -31.34, 179.02], [-0.029449, 0.706493, 0.698112, 0.112428], [0,0,0,0], [9E9, 9E9, 9E9, 9E9, 9E9, 9E9]];
	VAR robtarget Openhole_7328 := [[431.47, -29.27, 179.78], [-0.024808, 0.706671, 0.70072, 0.094826], [0,0,0,0], [9E9, 9E9, 9E9, 9E9, 9E9, 9E9]];
	VAR robtarget Openhole_7329 := [[437.75, -27.77, 180.57], [-0.008554, 0.707055, 0.70369, 0.069431], [0,0,0,0], [9E9, 9E9, 9E9, 9E9, 9E9, 9E9]];
	VAR robtarget Openhole_7330 := [[441.62, -26.84, 180.96], [0.001479, 0.707105, 0.705084, 0.053444], [0,0,0,0], [9E9, 9E9, 9E9, 9E9, 9E9, 9E9]];
	VAR robtarget Openhole_7331 := [[442.11, -26.73, 181], [0.002773, 0.707101, 0.705232, 0.051453], [0,0,0,0], [9E9, 9E9, 9E9, 9E9, 9E9, 9E9]];
	VAR robtarget Openhole_7332 := [[443.06, -26.45, 181.09], [0.005094, 0.707088, 0.705522, 0.04731], [0,0,0,0], [9E9, 9E9, 9E9, 9E9, 9E9, 9E9]];
	VAR robtarget Openhole_7333 := [[443.53, -26.29, 181.13], [0.006179, 0.70708, 0.705661, 0.045196], [0,0,0,0], [9E9, 9E9, 9E9, 9E9, 9E9, 9E9]];
	VAR robtarget Openhole_7334 := [[444.46, -25.91, 181.22], [0.008034, 0.707061, 0.705928, 0.040815], [0,0,0,0], [9E9, 9E9, 9E9, 9E9, 9E9, 9E9]];
	VAR robtarget Openhole_7335 := [[445.06, -25.46, 181.28], [0.008566, 0.707055, 0.706126, 0.037227], [0,0,0,0], [9E9, 9E9, 9E9, 9E9, 9E9, 9E9]];
	VAR robtarget Openhole_7336 := [[442.67, -23.11, 181.28], [-0.007588, 0.707066, 0.706119, 0.037365], [0,0,0,0], [9E9, 9E9, 9E9, 9E9, 9E9, 9E9]];
	VAR robtarget Openhole_7337 := [[442.05, -23.57, 181.22], [-0.008117, 0.70706, 0.705917, 0.040997], [0,0,0,0], [9E9, 9E9, 9E9, 9E9, 9E9, 9E9]];
	VAR robtarget Openhole_7338 := [[441.65, -23.86, 181.18], [-0.008503, 0.707056, 0.705777, 0.043337], [0,0,0,0], [9E9, 9E9, 9E9, 9E9, 9E9, 9E9]];
	VAR robtarget Openhole_7339 := [[441.23, -24.14, 181.14], [-0.008992, 0.70705, 0.705631, 0.045656], [0,0,0,0], [9E9, 9E9, 9E9, 9E9, 9E9, 9E9]];
	VAR robtarget Openhole_7340 := [[440.8, -24.39, 181.1], [-0.009606, 0.707042, 0.70548, 0.047942], [0,0,0,0], [9E9, 9E9, 9E9, 9E9, 9E9, 9E9]];
	VAR robtarget Openhole_7341 := [[439.91, -24.83, 181.01], [-0.011143, 0.707019, 0.705162, 0.052412], [0,0,0,0], [9E9, 9E9, 9E9, 9E9, 9E9, 9E9]];
	VAR robtarget Openhole_7342 := [[439.46, -25.04, 180.97], [-0.011968, 0.707006, 0.704994, 0.054624], [0,0,0,0], [9E9, 9E9, 9E9, 9E9, 9E9, 9E9]];
	VAR robtarget Openhole_7343 := [[438.55, -25.44, 180.87], [-0.013709, 0.706974, 0.704641, 0.058999], [0,0,0,0], [9E9, 9E9, 9E9, 9E9, 9E9, 9E9]];
	VAR robtarget Openhole_7344 := [[434.35, -26.98, 180.39], [-0.022762, 0.70674, 0.702795, 0.077967], [0,0,0,0], [9E9, 9E9, 9E9, 9E9, 9E9, 9E9]];
	VAR robtarget Openhole_7345 := [[432.92, -27.42, 180.22], [-0.026112, 0.706625, 0.702095, 0.084043], [0,0,0,0], [9E9, 9E9, 9E9, 9E9, 9E9, 9E9]];
	VAR robtarget Openhole_7346 := [[435.85, -24.75, 180.8], [-0.025192, 0.706658, 0.704057, 0.065603], [0,0,0,0], [9E9, 9E9, 9E9, 9E9, 9E9, 9E9]];
	VAR robtarget Openhole_7347 := [[437.63, -23.85, 181], [-0.02222, 0.706758, 0.704828, 0.056721], [0,0,0,0], [9E9, 9E9, 9E9, 9E9, 9E9, 9E9]];
	VAR robtarget Openhole_7348 := [[438.06, -23.61, 181.04], [-0.021544, 0.706779, 0.705006, 0.05447], [0,0,0,0], [9E9, 9E9, 9E9, 9E9, 9E9, 9E9]];
	VAR robtarget Openhole_7349 := [[439.34, -22.84, 181.17], [-0.019829, 0.706829, 0.705502, 0.04761], [0,0,0,0], [9E9, 9E9, 9E9, 9E9, 9E9, 9E9]];
	VAR robtarget Openhole_7350 := [[440.59, -22.01, 181.29], [-0.018411, 0.706867, 0.705937, 0.040652], [0,0,0,0], [9E9, 9E9, 9E9, 9E9, 9E9, 9E9]];
	VAR robtarget Openhole_7351 := [[441.01, -21.74, 181.32], [-0.017901, 0.70688, 0.706067, 0.038334], [0,0,0,0], [9E9, 9E9, 9E9, 9E9, 9E9, 9E9]];
	VAR robtarget Openhole_7352 := [[441.8, -21.35, 181.37], [-0.016545, 0.706913, 0.706272, 0.034359], [0,0,0,0], [9E9, 9E9, 9E9, 9E9, 9E9, 9E9]];
	VAR robtarget Openhole_7353 := [[438.17, -20.01, 181.44], [-0.033386, 0.706318, 0.705858, 0.042014], [0,0,0,0], [9E9, 9E9, 9E9, 9E9, 9E9, 9E9]];
	VAR robtarget Openhole_7354 := [[437.76, -20.3, 181.4], [-0.033794, 0.706299, 0.705715, 0.044342], [0,0,0,0], [9E9, 9E9, 9E9, 9E9, 9E9, 9E9]];
	VAR robtarget Openhole_7355 := [[436.96, -20.89, 181.32], [-0.034489, 0.706265, 0.705407, 0.049006], [0,0,0,0], [9E9, 9E9, 9E9, 9E9, 9E9, 9E9]];
	VAR robtarget Openhole_7356 := [[436.14, -21.45, 181.23], [-0.035354, 0.706222, 0.70507, 0.053626], [0,0,0,0], [9E9, 9E9, 9E9, 9E9, 9E9, 9E9]];
	VAR robtarget Openhole_7357 := [[435.72, -21.72, 181.19], [-0.035856, 0.706197, 0.704892, 0.055917], [0,0,0,0], [9E9, 9E9, 9E9, 9E9, 9E9, 9E9]];
	VAR robtarget Openhole_7358 := [[435.3, -21.98, 181.14], [-0.036399, 0.706169, 0.704708, 0.058193], [0,0,0,0], [9E9, 9E9, 9E9, 9E9, 9E9, 9E9]];
	VAR robtarget Openhole_7359 := [[434.43, -22.48, 181.05], [-0.03761, 0.706106, 0.704321, 0.062704], [0,0,0,0], [9E9, 9E9, 9E9, 9E9, 9E9, 9E9]];
	VAR robtarget Openhole_7360 := [[434, -22.72, 181], [-0.038283, 0.70607, 0.704119, 0.064934], [0,0,0,0], [9E9, 9E9, 9E9, 9E9, 9E9, 9E9]];
	VAR robtarget Openhole_7361 := [[433.55, -22.94, 180.95], [-0.039017, 0.70603, 0.703912, 0.06714], [0,0,0,0], [9E9, 9E9, 9E9, 9E9, 9E9, 9E9]];
	VAR robtarget Openhole_7362 := [[432.65, -23.37, 180.84], [-0.04061, 0.70594, 0.703483, 0.071497], [0,0,0,0], [9E9, 9E9, 9E9, 9E9, 9E9, 9E9]];
	VAR robtarget Openhole_7363 := [[432.19, -23.56, 180.79], [-0.04149, 0.705888, 0.703262, 0.073635], [0,0,0,0], [9E9, 9E9, 9E9, 9E9, 9E9, 9E9]];
	VAR robtarget Openhole_7364 := [[431.73, -23.75, 180.74], [-0.04241, 0.705834, 0.703037, 0.075753], [0,0,0,0], [9E9, 9E9, 9E9, 9E9, 9E9, 9E9]];
	VAR robtarget Openhole_7365 := [[430.8, -24.09, 180.64], [-0.044368, 0.705713, 0.702576, 0.079922], [0,0,0,0], [9E9, 9E9, 9E9, 9E9, 9E9, 9E9]];
	VAR robtarget Openhole_7366 := [[430.33, -24.25, 180.59], [-0.045419, 0.705647, 0.70234, 0.081964], [0,0,0,0], [9E9, 9E9, 9E9, 9E9, 9E9, 9E9]];
	VAR robtarget Openhole_7367 := [[427.45, -25.03, 180.28], [-0.052377, 0.705164, 0.700864, 0.093752], [0,0,0,0], [9E9, 9E9, 9E9, 9E9, 9E9, 9E9]];
	VAR robtarget Openhole_7368 := [[426.96, -25.13, 180.23], [-0.053633, 0.70507, 0.700609, 0.09564], [0,0,0,0], [9E9, 9E9, 9E9, 9E9, 9E9, 9E9]];
	VAR robtarget Openhole_7369 := [[425, -25.46, 180.03], [-0.058973, 0.704643, 0.699577, 0.102916], [0,0,0,0], [9E9, 9E9, 9E9, 9E9, 9E9, 9E9]];
	VAR robtarget Openhole_7370 := [[421.04, -25.86, 179.68], [-0.070562, 0.703577, 0.697451, 0.116456], [0,0,0,0], [9E9, 9E9, 9E9, 9E9, 9E9, 9E9]];
	VAR robtarget Openhole_7371 := [[416.05, -25.98, 179.31], [-0.086024, 0.701855, 0.694707, 0.13184], [0,0,0,0], [9E9, 9E9, 9E9, 9E9, 9E9, 9E9]];
	VAR robtarget Openhole_7372 := [[415.55, -25.97, 179.28], [-0.087602, 0.701659, 0.694429, 0.133301], [0,0,0,0], [9E9, 9E9, 9E9, 9E9, 9E9, 9E9]];
	VAR robtarget Openhole_7373 := [[401.58, -25.68, 178.48], [-0.130373, 0.694984, 0.685999, 0.171479], [0,0,0,0], [9E9, 9E9, 9E9, 9E9, 9E9, 9E9]];
	VAR robtarget Openhole_7374 := [[401.08, -25.68, 178.45], [-0.131791, 0.694717, 0.685669, 0.172795], [0,0,0,0], [9E9, 9E9, 9E9, 9E9, 9E9, 9E9]];
	VAR robtarget Openhole_7375 := [[395.6, -25.83, 178.02], [-0.14655, 0.691754, 0.681846, 0.187313], [0,0,0,0], [9E9, 9E9, 9E9, 9E9, 9E9, 9E9]];
	VAR robtarget Openhole_7376 := [[395.1, -25.86, 177.97], [-0.147808, 0.691486, 0.68148, 0.188639], [0,0,0,0], [9E9, 9E9, 9E9, 9E9, 9E9, 9E9]];
	VAR robtarget Openhole_7377 := [[394.34, -25.89, 177.91], [-0.149812, 0.691055, 0.680932, 0.19061], [0,0,0,0], [9E9, 9E9, 9E9, 9E9, 9E9, 9E9]];
	VAR robtarget Openhole_7378 := [[389.33, -25.89, 177.58], [-0.162982, 0.688068, 0.677437, 0.202679], [0,0,0,0], [9E9, 9E9, 9E9, 9E9, 9E9, 9E9]];
	VAR robtarget Openhole_7379 := [[362.33, -25.89, 177.66], [-0.183051, 0.683002, 0.683002, 0.183051], [0,0,0,0], [9E9, 9E9, 9E9, 9E9, 9E9, 9E9]];
	VAR robtarget Openhole_7380 := [[362.34, -25.1, 178.12], [-0.183051, 0.683002, 0.683002, 0.183051], [0,0,0,0], [9E9, 9E9, 9E9, 9E9, 9E9, 9E9]];
	VAR robtarget Openhole_7381 := [[389.34, -25.1, 178.03], [-0.165233, 0.687531, 0.678095, 0.200467], [0,0,0,0], [9E9, 9E9, 9E9, 9E9, 9E9, 9E9]];
	VAR robtarget Openhole_7382 := [[394.34, -25.1, 178.33], [-0.152119, 0.69055, 0.681563, 0.188342], [0,0,0,0], [9E9, 9E9, 9E9, 9E9, 9E9, 9E9]];
	VAR robtarget Openhole_7383 := [[395.22, -25.08, 178.39], [-0.149805, 0.691056, 0.682187, 0.186066], [0,0,0,0], [9E9, 9E9, 9E9, 9E9, 9E9, 9E9]];
	VAR robtarget Openhole_7384 := [[400.7, -24.87, 178.81], [-0.135307, 0.69404, 0.686022, 0.171387], [0,0,0,0], [9E9, 9E9, 9E9, 9E9, 9E9, 9E9]];
	VAR robtarget Openhole_7385 := [[402.2, -24.86, 178.89], [-0.131095, 0.694848, 0.687009, 0.167388], [0,0,0,0], [9E9, 9E9, 9E9, 9E9, 9E9, 9E9]];
	VAR robtarget Openhole_7386 := [[402.7, -24.86, 178.92], [-0.129665, 0.695117, 0.687332, 0.166057], [0,0,0,0], [9E9, 9E9, 9E9, 9E9, 9E9, 9E9]];
	VAR robtarget Openhole_7387 := [[416.18, -25.08, 179.61], [-0.088501, 0.701547, 0.695309, 0.128631], [0,0,0,0], [9E9, 9E9, 9E9, 9E9, 9E9, 9E9]];
	VAR robtarget Openhole_7388 := [[416.68, -25.08, 179.64], [-0.08694, 0.701742, 0.695583, 0.12714], [0,0,0,0], [9E9, 9E9, 9E9, 9E9, 9E9, 9E9]];
	VAR robtarget Openhole_7389 := [[422.16, -24.91, 180], [-0.070038, 0.70363, 0.698509, 0.109931], [0,0,0,0], [9E9, 9E9, 9E9, 9E9, 9E9, 9E9]];
	VAR robtarget Openhole_7390 := [[424.15, -24.72, 180.16], [-0.064212, 0.704185, 0.699541, 0.10316], [0,0,0,0], [9E9, 9E9, 9E9, 9E9, 9E9, 9E9]];
	VAR robtarget Openhole_7391 := [[425.14, -24.59, 180.24], [-0.0614, 0.704436, 0.700049, 0.099654], [0,0,0,0], [9E9, 9E9, 9E9, 9E9, 9E9, 9E9]];
	VAR robtarget Openhole_7392 := [[426.61, -24.36, 180.37], [-0.057332, 0.704779, 0.7008, 0.094233], [0,0,0,0], [9E9, 9E9, 9E9, 9E9, 9E9, 9E9]];
	VAR robtarget Openhole_7393 := [[427.1, -24.27, 180.42], [-0.056037, 0.704883, 0.701047, 0.092372], [0,0,0,0], [9E9, 9E9, 9E9, 9E9, 9E9, 9E9]];
	VAR robtarget Openhole_7394 := [[428.07, -24.05, 180.51], [-0.053544, 0.705077, 0.701538, 0.088568], [0,0,0,0], [9E9, 9E9, 9E9, 9E9, 9E9, 9E9]];
	VAR robtarget Openhole_7395 := [[429.52, -23.69, 180.65], [-0.049965, 0.705339, 0.702252, 0.08272], [0,0,0,0], [9E9, 9E9, 9E9, 9E9, 9E9, 9E9]];
	VAR robtarget Openhole_7396 := [[430.48, -23.42, 180.74], [-0.0477, 0.705496, 0.702711, 0.078724], [0,0,0,0], [9E9, 9E9, 9E9, 9E9, 9E9, 9E9]];
	VAR robtarget Openhole_7397 := [[428.63, -22.36, 180.88], [-0.057359, 0.704777, 0.70243, 0.081189], [0,0,0,0], [9E9, 9E9, 9E9, 9E9, 9E9, 9E9]];
	VAR robtarget Openhole_7398 := [[428.14, -22.45, 180.84], [-0.058653, 0.70467, 0.70221, 0.083077], [0,0,0,0], [9E9, 9E9, 9E9, 9E9, 9E9, 9E9]];
	VAR robtarget Openhole_7399 := [[425.18, -22.88, 180.64], [-0.066922, 0.703933, 0.700841, 0.093923], [0,0,0,0], [9E9, 9E9, 9E9, 9E9, 9E9, 9E9]];
	VAR robtarget Openhole_7400 := [[420.7, -23.18, 180.4], [-0.080399, 0.702521, 0.698676, 0.108867], [0,0,0,0], [9E9, 9E9, 9E9, 9E9, 9E9, 9E9]];
	VAR robtarget Openhole_7401 := [[418.2, -23.21, 180.29], [-0.08821, 0.701583, 0.697427, 0.1166], [0,0,0,0], [9E9, 9E9, 9E9, 9E9, 9E9, 9E9]];
	VAR robtarget Openhole_7402 := [[417.7, -23.21, 180.27], [-0.089781, 0.701384, 0.697173, 0.118111], [0,0,0,0], [9E9, 9E9, 9E9, 9E9, 9E9, 9E9]];
	VAR robtarget Openhole_7403 := [[417.2, -23.21, 180.25], [-0.091344, 0.701182, 0.696915, 0.119622], [0,0,0,0], [9E9, 9E9, 9E9, 9E9, 9E9, 9E9]];
	VAR robtarget Openhole_7404 := [[416.7, -23.21, 180.23], [-0.092917, 0.700975, 0.696658, 0.121112], [0,0,0,0], [9E9, 9E9, 9E9, 9E9, 9E9, 9E9]];
	VAR robtarget Openhole_7405 := [[404.71, -23.06, 179.81], [-0.129425, 0.695161, 0.689874, 0.155158], [0,0,0,0], [9E9, 9E9, 9E9, 9E9, 9E9, 9E9]];
	VAR robtarget Openhole_7406 := [[404.21, -23.06, 179.79], [-0.13086, 0.694893, 0.689564, 0.15653], [0,0,0,0], [9E9, 9E9, 9E9, 9E9, 9E9, 9E9]];
	VAR robtarget Openhole_7407 := [[397.22, -23.22, 179.44], [-0.149897, 0.691036, 0.684961, 0.175582], [0,0,0,0], [9E9, 9E9, 9E9, 9E9, 9E9, 9E9]];
	VAR robtarget Openhole_7408 := [[395.23, -23.34, 179.3], [-0.154924, 0.689927, 0.683548, 0.181002], [0,0,0,0], [9E9, 9E9, 9E9, 9E9, 9E9, 9E9]];
	VAR robtarget Openhole_7409 := [[394.34, -23.36, 179.25], [-0.157217, 0.689408, 0.682931, 0.183317], [0,0,0,0], [9E9, 9E9, 9E9, 9E9, 9E9, 9E9]];
	VAR robtarget Openhole_7410 := [[389.34, -23.36, 179.04], [-0.170205, 0.686316, 0.679524, 0.195567], [0,0,0,0], [9E9, 9E9, 9E9, 9E9, 9E9, 9E9]];
	VAR robtarget Openhole_7411 := [[362.34, -23.36, 179.12], [-0.183051, 0.683002, 0.683002, 0.183051], [0,0,0,0], [9E9, 9E9, 9E9, 9E9, 9E9, 9E9]];
	VAR robtarget Openhole_7412 := [[362.34, -22.46, 179.64], [-0.183051, 0.683002, 0.683002, 0.183051], [0,0,0,0], [9E9, 9E9, 9E9, 9E9, 9E9, 9E9]];
	VAR robtarget Openhole_7413 := [[389.34, -22.46, 179.56], [-0.172787, 0.685671, 0.680254, 0.193016], [0,0,0,0], [9E9, 9E9, 9E9, 9E9, 9E9, 9E9]];
	VAR robtarget Openhole_7414 := [[394.34, -22.46, 179.72], [-0.159864, 0.688799, 0.683628, 0.180701], [0,0,0,0], [9E9, 9E9, 9E9, 9E9, 9E9, 9E9]];
	VAR robtarget Openhole_7415 := [[395.12, -22.43, 179.76], [-0.157883, 0.689255, 0.684169, 0.178641], [0,0,0,0], [9E9, 9E9, 9E9, 9E9, 9E9, 9E9]];
	VAR robtarget Openhole_7416 := [[401.61, -22.16, 180.1], [-0.140989, 0.692909, 0.688561, 0.160883], [0,0,0,0], [9E9, 9E9, 9E9, 9E9, 9E9, 9E9]];
	VAR robtarget Openhole_7417 := [[405.6, -22.12, 180.24], [-0.129736, 0.695103, 0.691051, 0.149828], [0,0,0,0], [9E9, 9E9, 9E9, 9E9, 9E9, 9E9]];
	VAR robtarget Openhole_7418 := [[406.1, -22.12, 180.25], [-0.128289, 0.695372, 0.691351, 0.148437], [0,0,0,0], [9E9, 9E9, 9E9, 9E9, 9E9, 9E9]];
	VAR robtarget Openhole_7419 := [[418.1, -22.26, 180.57], [-0.091591, 0.70115, 0.697877, 0.113877], [0,0,0,0], [9E9, 9E9, 9E9, 9E9, 9E9, 9E9]];
	VAR robtarget Openhole_7420 := [[418.6, -22.26, 180.58], [-0.090022, 0.701353, 0.698124, 0.112354], [0,0,0,0], [9E9, 9E9, 9E9, 9E9, 9E9, 9E9]];
	VAR robtarget Openhole_7421 := [[423.09, -22.18, 180.74], [-0.075984, 0.703012, 0.700256, 0.09819], [0,0,0,0], [9E9, 9E9, 9E9, 9E9, 9E9, 9E9]];
	VAR robtarget Openhole_7422 := [[427.57, -21.76, 180.97], [-0.062837, 0.704309, 0.702262, 0.082636], [0,0,0,0], [9E9, 9E9, 9E9, 9E9, 9E9, 9E9]];
	VAR robtarget Openhole_7423 := [[428.06, -21.68, 181], [-0.061471, 0.70443, 0.702475, 0.080802], [0,0,0,0], [9E9, 9E9, 9E9, 9E9, 9E9, 9E9]];
	VAR robtarget Openhole_7424 := [[429.04, -21.5, 181.06], [-0.058839, 0.704654, 0.702897, 0.077044], [0,0,0,0], [9E9, 9E9, 9E9, 9E9, 9E9, 9E9]];
	VAR robtarget Openhole_7425 := [[430.02, -21.29, 181.12], [-0.05635, 0.704858, 0.703311, 0.073171], [0,0,0,0], [9E9, 9E9, 9E9, 9E9, 9E9, 9E9]];
	VAR robtarget Openhole_7426 := [[432.43, -20.64, 181.28], [-0.050521, 0.7053, 0.70428, 0.063161], [0,0,0,0], [9E9, 9E9, 9E9, 9E9, 9E9, 9E9]];
	VAR robtarget Openhole_7427 := [[433.85, -20.18, 181.37], [-0.047323, 0.705521, 0.704811, 0.056933], [0,0,0,0], [9E9, 9E9, 9E9, 9E9, 9E9, 9E9]];
	VAR robtarget Openhole_7428 := [[434.32, -20.01, 181.4], [-0.046344, 0.705586, 0.70498, 0.054807], [0,0,0,0], [9E9, 9E9, 9E9, 9E9, 9E9, 9E9]];
	VAR robtarget Openhole_7429 := [[434.78, -19.82, 181.43], [-0.045438, 0.705645, 0.705144, 0.052645], [0,0,0,0], [9E9, 9E9, 9E9, 9E9, 9E9, 9E9]];
	VAR robtarget Openhole_7430 := [[435.69, -19.42, 181.49], [-0.043736, 0.705753, 0.705458, 0.048265], [0,0,0,0], [9E9, 9E9, 9E9, 9E9, 9E9, 9E9]];
	VAR robtarget Openhole_7431 := [[436.63, -19.07, 181.54], [-0.04176, 0.705873, 0.705737, 0.043984], [0,0,0,0], [9E9, 9E9, 9E9, 9E9, 9E9, 9E9]];
	VAR robtarget Openhole_7432 := [[437.08, -18.86, 181.56], [-0.040967, 0.705919, 0.705873, 0.041759], [0,0,0,0], [9E9, 9E9, 9E9, 9E9, 9E9, 9E9]];
	VAR robtarget Openhole_7433 := [[436.54, -17.57, 181.72], [-0.047139, 0.705534, 0.706016, 0.039266], [0,0,0,0], [9E9, 9E9, 9E9, 9E9, 9E9, 9E9]];
	VAR robtarget Openhole_7434 := [[435.54, -17.56, 181.74], [-0.050514, 0.7053, 0.705824, 0.042573], [0,0,0,0], [9E9, 9E9, 9E9, 9E9, 9E9, 9E9]];
	VAR robtarget Openhole_7435 := [[435.04, -17.58, 181.74], [-0.05212, 0.705183, 0.705718, 0.0443], [0,0,0,0], [9E9, 9E9, 9E9, 9E9, 9E9, 9E9]];
	VAR robtarget Openhole_7436 := [[434.54, -17.58, 181.75], [-0.05379, 0.705058, 0.705612, 0.045959], [0,0,0,0], [9E9, 9E9, 9E9, 9E9, 9E9, 9E9]];
	VAR robtarget Openhole_7437 := [[434.04, -17.59, 181.75], [-0.055442, 0.70493, 0.705501, 0.047631], [0,0,0,0], [9E9, 9E9, 9E9, 9E9, 9E9, 9E9]];
	VAR robtarget Openhole_7438 := [[433.54, -17.58, 181.76], [-0.057131, 0.704795, 0.705389, 0.049261], [0,0,0,0], [9E9, 9E9, 9E9, 9E9, 9E9, 9E9]];
	VAR robtarget Openhole_7439 := [[433.04, -17.58, 181.77], [-0.058769, 0.70466, 0.70527, 0.050937], [0,0,0,0], [9E9, 9E9, 9E9, 9E9, 9E9, 9E9]];
	VAR robtarget Openhole_7440 := [[432.54, -17.58, 181.77], [-0.060429, 0.70452, 0.705149, 0.052585], [0,0,0,0], [9E9, 9E9, 9E9, 9E9, 9E9, 9E9]];
	VAR robtarget Openhole_7441 := [[418.04, -17.3, 182.06], [-0.107819, 0.698838, 0.700267, 0.098114], [0,0,0,0], [9E9, 9E9, 9E9, 9E9, 9E9, 9E9]];
	VAR robtarget Openhole_7442 := [[408.55, -17.2, 182.26], [-0.136524, 0.693802, 0.695737, 0.126293], [0,0,0,0], [9E9, 9E9, 9E9, 9E9, 9E9, 9E9]];
	VAR robtarget Openhole_7443 := [[408.05, -17.2, 182.27], [-0.137961, 0.693518, 0.695471, 0.127748], [0,0,0,0], [9E9, 9E9, 9E9, 9E9, 9E9, 9E9]];
	VAR robtarget Openhole_7444 := [[398.55, -17.4, 182.34], [-0.163695, 0.687898, 0.689939, 0.15487], [0,0,0,0], [9E9, 9E9, 9E9, 9E9, 9E9, 9E9]];
	VAR robtarget Openhole_7445 := [[394.35, -17.6, 182.3], [-0.174103, 0.685338, 0.687215, 0.166541], [0,0,0,0], [9E9, 9E9, 9E9, 9E9, 9E9, 9E9]];
	VAR robtarget Openhole_7446 := [[362.35, -17.6, 182.45], [-0.183051, 0.683002, 0.683002, 0.183051], [0,0,0,0], [9E9, 9E9, 9E9, 9E9, 9E9, 9E9]];
	VAR robtarget Openhole_7447 := [[362.35, -18.56, 181.9], [-0.183051, 0.683002, 0.683002, 0.183051], [0,0,0,0], [9E9, 9E9, 9E9, 9E9, 9E9, 9E9]];
	VAR robtarget Openhole_7448 := [[389.35, -18.56, 181.81], [-0.183933, 0.682765, 0.683299, 0.181941], [0,0,0,0], [9E9, 9E9, 9E9, 9E9, 9E9, 9E9]];
	VAR robtarget Openhole_7449 := [[394.35, -18.56, 181.79], [-0.171295, 0.686045, 0.686529, 0.169345], [0,0,0,0], [9E9, 9E9, 9E9, 9E9, 9E9, 9E9]];
	VAR robtarget Openhole_7450 := [[402.43, -18.22, 181.9], [-0.150656, 0.690871, 0.691706, 0.146773], [0,0,0,0], [9E9, 9E9, 9E9, 9E9, 9E9, 9E9]];
	VAR robtarget Openhole_7451 := [[408.43, -18.16, 181.88], [-0.133867, 0.694319, 0.695128, 0.129602], [0,0,0,0], [9E9, 9E9, 9E9, 9E9, 9E9, 9E9]];
	VAR robtarget Openhole_7452 := [[408.93, -18.16, 181.88], [-0.132411, 0.694599, 0.695396, 0.128158], [0,0,0,0], [9E9, 9E9, 9E9, 9E9, 9E9, 9E9]];
	VAR robtarget Openhole_7453 := [[426.43, -18.45, 181.67], [-0.077559, 0.70284, 0.703078, 0.075376], [0,0,0,0], [9E9, 9E9, 9E9, 9E9, 9E9, 9E9]];
	VAR robtarget Openhole_7454 := [[426.93, -18.44, 181.67], [-0.075946, 0.703017, 0.703249, 0.07376], [0,0,0,0], [9E9, 9E9, 9E9, 9E9, 9E9, 9E9]];
	VAR robtarget Openhole_7455 := [[430.43, -18.38, 181.66], [-0.064713, 0.704139, 0.704366, 0.062192], [0,0,0,0], [9E9, 9E9, 9E9, 9E9, 9E9, 9E9]];
	VAR robtarget Openhole_7456 := [[431.43, -18.38, 181.65], [-0.061414, 0.704435, 0.704648, 0.058918], [0,0,0,0], [9E9, 9E9, 9E9, 9E9, 9E9, 9E9]];
	VAR robtarget Openhole_7457 := [[431.93, -18.36, 181.65], [-0.059862, 0.704568, 0.704791, 0.05718], [0,0,0,0], [9E9, 9E9, 9E9, 9E9, 9E9, 9E9]];
	VAR robtarget Openhole_7458 := [[433.09, -19.64, 181.45], [-0.051674, 0.705216, 0.704755, 0.057626], [0,0,0,0], [9E9, 9E9, 9E9, 9E9, 9E9, 9E9]];
	VAR robtarget Openhole_7459 := [[431.14, -20.07, 181.36], [-0.0567, 0.70483, 0.704069, 0.065469], [0,0,0,0], [9E9, 9E9, 9E9, 9E9, 9E9, 9E9]];
	VAR robtarget Openhole_7460 := [[429.67, -20.35, 181.29], [-0.060623, 0.704503, 0.703513, 0.071197], [0,0,0,0], [9E9, 9E9, 9E9, 9E9, 9E9, 9E9]];
	VAR robtarget Openhole_7461 := [[429.18, -20.43, 181.27], [-0.06199, 0.704384, 0.703323, 0.073053], [0,0,0,0], [9E9, 9E9, 9E9, 9E9, 9E9, 9E9]];
	VAR robtarget Openhole_7462 := [[428.18, -20.56, 181.23], [-0.064817, 0.70413, 0.702937, 0.076681], [0,0,0,0], [9E9, 9E9, 9E9, 9E9, 9E9, 9E9]];
	VAR robtarget Openhole_7463 := [[426.19, -20.74, 181.16], [-0.070715, 0.703562, 0.70214, 0.083666], [0,0,0,0], [9E9, 9E9, 9E9, 9E9, 9E9, 9E9]];
	VAR robtarget Openhole_7464 := [[425.2, -20.8, 181.13], [-0.073737, 0.703252, 0.701727, 0.087058], [0,0,0,0], [9E9, 9E9, 9E9, 9E9, 9E9, 9E9]];
	VAR robtarget Openhole_7465 := [[421.2, -20.9, 181.03], [-0.086251, 0.701827, 0.700009, 0.099934], [0,0,0,0], [9E9, 9E9, 9E9, 9E9, 9E9, 9E9]];
	VAR robtarget Openhole_7466 := [[420.7, -20.89, 181.03], [-0.087843, 0.701629, 0.699787, 0.10148], [0,0,0,0], [9E9, 9E9, 9E9, 9E9, 9E9, 9E9]];
	VAR robtarget Openhole_7467 := [[406.7, -20.73, 180.84], [-0.13088, 0.694889, 0.692604, 0.142479], [0,0,0,0], [9E9, 9E9, 9E9, 9E9, 9E9, 9E9]];
	VAR robtarget Openhole_7468 := [[406.2, -20.73, 180.84], [-0.132321, 0.694616, 0.692312, 0.143891], [0,0,0,0], [9E9, 9E9, 9E9, 9E9, 9E9, 9E9]];
	VAR robtarget Openhole_7469 := [[398.21, -20.89, 180.62], [-0.154176, 0.690094, 0.68731, 0.166147], [0,0,0,0], [9E9, 9E9, 9E9, 9E9, 9E9, 9E9]];
	VAR robtarget Openhole_7470 := [[395.22, -21.06, 180.48], [-0.161682, 0.688374, 0.685262, 0.174403], [0,0,0,0], [9E9, 9E9, 9E9, 9E9, 9E9, 9E9]];
	VAR robtarget Openhole_7471 := [[394.34, -21.09, 180.45], [-0.163882, 0.687854, 0.684668, 0.176719], [0,0,0,0], [9E9, 9E9, 9E9, 9E9, 9E9, 9E9]];
	VAR robtarget Openhole_7472 := [[389.34, -21.09, 180.35], [-0.176705, 0.684672, 0.681343, 0.189133], [0,0,0,0], [9E9, 9E9, 9E9, 9E9, 9E9, 9E9]];
	VAR robtarget Openhole_7473 := [[362.34, -21.09, 180.43], [-0.183051, 0.683002, 0.683002, 0.183051], [0,0,0,0], [9E9, 9E9, 9E9, 9E9, 9E9, 9E9]];
	VAR robtarget Openhole_7474 := [[362.35, -15.88, 183.45], [-0.183051, 0.683002, 0.683002, 0.183051], [0,0,0,0], [9E9, 9E9, 9E9, 9E9, 9E9, 9E9]];
	VAR robtarget Openhole_7475 := [[389.35, -15.88, 183.36], [-0.191566, 0.680663, 0.685288, 0.174301], [0,0,0,0], [9E9, 9E9, 9E9, 9E9, 9E9, 9E9]];
	VAR robtarget Openhole_7476 := [[394.35, -15.88, 183.21], [-0.179124, 0.684043, 0.688414, 0.161513], [0,0,0,0], [9E9, 9E9, 9E9, 9E9, 9E9, 9E9]];
	VAR robtarget Openhole_7477 := [[402.84, -15.53, 183.11], [-0.157702, 0.689297, 0.693616, 0.137466], [0,0,0,0], [9E9, 9E9, 9E9, 9E9, 9E9, 9E9]];
	VAR robtarget Openhole_7478 := [[411.34, -15.42, 182.86], [-0.13397, 0.6943, 0.698099, 0.112509], [0,0,0,0], [9E9, 9E9, 9E9, 9E9, 9E9, 9E9]];
	VAR robtarget Openhole_7479 := [[411.84, -15.42, 182.84], [-0.132504, 0.694581, 0.698338, 0.111015], [0,0,0,0], [9E9, 9E9, 9E9, 9E9, 9E9, 9E9]];
	VAR robtarget Openhole_7480 := [[425.83, -15.62, 182.31], [-0.088836, 0.701504, 0.703829, 0.068009], [0,0,0,0], [9E9, 9E9, 9E9, 9E9, 9E9, 9E9]];
	VAR robtarget Openhole_7481 := [[433.81, -16, 181.99], [-0.061529, 0.704425, 0.705794, 0.043071], [0,0,0,0], [9E9, 9E9, 9E9, 9E9, 9E9, 9E9]];
	VAR robtarget Openhole_7482 := [[434.81, -16.09, 181.95], [-0.057907, 0.704732, 0.70597, 0.040078], [0,0,0,0], [9E9, 9E9, 9E9, 9E9, 9E9, 9E9]];
	VAR robtarget Openhole_7483 := [[435.3, -16.15, 181.93], [-0.056057, 0.704881, 0.706051, 0.038621], [0,0,0,0], [9E9, 9E9, 9E9, 9E9, 9E9, 9E9]];
	VAR robtarget Openhole_7484 := [[438.22, -12.1, 182.28], [-0.060002, 0.704556, 0.706943, 0.015211], [0,0,0,0], [9E9, 9E9, 9E9, 9E9, 9E9, 9E9]];
	VAR robtarget Openhole_7485 := [[439.21, -12.15, 182.21], [-0.056484, 0.704847, 0.707004, 0.012032], [0,0,0,0], [9E9, 9E9, 9E9, 9E9, 9E9, 9E9]];
	VAR robtarget Openhole_7486 := [[440.21, -12.22, 182.14], [-0.052898, 0.705125, 0.707051, 0.008914], [0,0,0,0], [9E9, 9E9, 9E9, 9E9, 9E9, 9E9]];
	VAR robtarget Openhole_7487 := [[441.7, -12.31, 182.04], [-0.047577, 0.705504, 0.707095, 0.004144], [0,0,0,0], [9E9, 9E9, 9E9, 9E9, 9E9, 9E9]];
	VAR robtarget Openhole_7488 := [[442.2, -12.35, 182], [-0.045768, 0.705624, 0.707102, 0.002588], [0,0,0,0], [9E9, 9E9, 9E9, 9E9, 9E9, 9E9]];
	VAR robtarget Openhole_7489 := [[443.19, -12.46, 181.93], [-0.042043, 0.705856, 0.707107, -0.000404], [0,0,0,0], [9E9, 9E9, 9E9, 9E9, 9E9, 9E9]];
	VAR robtarget Openhole_7490 := [[443.92, -12.82, 181.87], [-0.038338, 0.706067, 0.707105, -0.001664], [0,0,0,0], [9E9, 9E9, 9E9, 9E9, 9E9, 9E9]];
	VAR robtarget Openhole_7491 := [[455.86, -14.06, 181.23], [0.006581, 0.707076, 0.706089, -0.037933], [0,0,0,0], [9E9, 9E9, 9E9, 9E9, 9E9, 9E9]];
	VAR robtarget Openhole_7492 := [[456.33, -13.69, 181.18], [0.006916, 0.707073, 0.705931, -0.040761], [0,0,0,0], [9E9, 9E9, 9E9, 9E9, 9E9, 9E9]];
	VAR robtarget Openhole_7493 := [[456.74, -13.4, 181.14], [0.007299, 0.707069, 0.705792, -0.043103], [0,0,0,0], [9E9, 9E9, 9E9, 9E9, 9E9, 9E9]];
	VAR robtarget Openhole_7494 := [[457.16, -13.13, 181.1], [0.007814, 0.707064, 0.705647, -0.045418], [0,0,0,0], [9E9, 9E9, 9E9, 9E9, 9E9, 9E9]];
	VAR robtarget Openhole_7495 := [[457.59, -12.89, 181.05], [0.008505, 0.707056, 0.705497, -0.047684], [0,0,0,0], [9E9, 9E9, 9E9, 9E9, 9E9, 9E9]];
	VAR robtarget Openhole_7496 := [[458.49, -12.46, 180.96], [0.010098, 0.707035, 0.705182, -0.052139], [0,0,0,0], [9E9, 9E9, 9E9, 9E9, 9E9, 9E9]];
	VAR robtarget Openhole_7497 := [[459.4, -12.06, 180.87], [0.011853, 0.707007, 0.704844, -0.056522], [0,0,0,0], [9E9, 9E9, 9E9, 9E9, 9E9, 9E9]];
	VAR robtarget Openhole_7498 := [[461.73, -11.18, 180.61], [0.016747, 0.706908, 0.703906, -0.0672], [0,0,0,0], [9E9, 9E9, 9E9, 9E9, 9E9, 9E9]];
	VAR robtarget Openhole_7499 := [[464.08, -10.39, 180.32], [0.022077, 0.706762, 0.70284, -0.077566], [0,0,0,0], [9E9, 9E9, 9E9, 9E9, 9E9, 9E9]];
	VAR robtarget Openhole_7500 := [[465.51, -9.96, 180.13], [0.025447, 0.706649, 0.702143, -0.083639], [0,0,0,0], [9E9, 9E9, 9E9, 9E9, 9E9, 9E9]];
	VAR robtarget Openhole_7501 := [[468.4, -7.76, 179.47], [0.02786, 0.706558, 0.69997, -0.100209], [0,0,0,0], [9E9, 9E9, 9E9, 9E9, 9E9, 9E9]];
	VAR robtarget Openhole_7502 := [[460.66, -9.48, 180.5], [0.007387, 0.707068, 0.703699, -0.069334], [0,0,0,0], [9E9, 9E9, 9E9, 9E9, 9E9, 9E9]];
	VAR robtarget Openhole_7503 := [[457.75, -10.16, 180.82], [-0.000181, 0.707107, 0.704774, -0.057384], [0,0,0,0], [9E9, 9E9, 9E9, 9E9, 9E9, 9E9]];
	VAR robtarget Openhole_7504 := [[456.79, -10.4, 180.92], [-0.002689, 0.707102, 0.70509, -0.053363], [0,0,0,0], [9E9, 9E9, 9E9, 9E9, 9E9, 9E9]];
	VAR robtarget Openhole_7505 := [[456.31, -10.53, 180.97], [-0.003897, 0.707096, 0.705242, -0.051322], [0,0,0,0], [9E9, 9E9, 9E9, 9E9, 9E9, 9E9]];
	VAR robtarget Openhole_7506 := [[455.82, -10.65, 181.02], [-0.005143, 0.707088, 0.705386, -0.049299], [0,0,0,0], [9E9, 9E9, 9E9, 9E9, 9E9, 9E9]];
	VAR robtarget Openhole_7507 := [[454.86, -10.92, 181.11], [-0.007501, 0.707067, 0.705663, -0.045168], [0,0,0,0], [9E9, 9E9, 9E9, 9E9, 9E9, 9E9]];
	VAR robtarget Openhole_7508 := [[454.39, -11.08, 181.16], [-0.008568, 0.707055, 0.705796, -0.043041], [0,0,0,0], [9E9, 9E9, 9E9, 9E9, 9E9, 9E9]];
	VAR robtarget Openhole_7509 := [[453.93, -11.26, 181.2], [-0.009508, 0.707043, 0.705926, -0.040855], [0,0,0,0], [9E9, 9E9, 9E9, 9E9, 9E9, 9E9]];
	VAR robtarget Openhole_7510 := [[453.31, -11.75, 181.26], [-0.010008, 0.707036, 0.706132, -0.03711], [0,0,0,0], [9E9, 9E9, 9E9, 9E9, 9E9, 9E9]];
	VAR robtarget Openhole_7511 := [[446.72, -11.14, 181.74], [-0.034528, 0.706263, 0.706907, -0.016826], [0,0,0,0], [9E9, 9E9, 9E9, 9E9, 9E9, 9E9]];
	VAR robtarget Openhole_7512 := [[446.16, -10.86, 181.79], [-0.037408, 0.706117, 0.706928, -0.015899], [0,0,0,0], [9E9, 9E9, 9E9, 9E9, 9E9, 9E9]];
	VAR robtarget Openhole_7513 := [[445.18, -10.67, 181.88], [-0.041354, 0.705896, 0.706984, -0.013188], [0,0,0,0], [9E9, 9E9, 9E9, 9E9, 9E9, 9E9]];
	VAR robtarget Openhole_7514 := [[444.69, -10.59, 181.92], [-0.043295, 0.70578, 0.707008, -0.011792], [0,0,0,0], [9E9, 9E9, 9E9, 9E9, 9E9, 9E9]];
	VAR robtarget Openhole_7515 := [[444.19, -10.54, 181.96], [-0.045149, 0.705664, 0.707032, -0.010283], [0,0,0,0], [9E9, 9E9, 9E9, 9E9, 9E9, 9E9]];
	VAR robtarget Openhole_7516 := [[443.7, -10.51, 182], [-0.04693, 0.705548, 0.707053, -0.008691], [0,0,0,0], [9E9, 9E9, 9E9, 9E9, 9E9, 9E9]];
	VAR robtarget Openhole_7517 := [[442.7, -10.49, 182.09], [-0.050364, 0.705311, 0.707086, -0.005373], [0,0,0,0], [9E9, 9E9, 9E9, 9E9, 9E9, 9E9]];
	VAR robtarget Openhole_7518 := [[439.21, -10.53, 182.37], [-0.061945, 0.704388, 0.707076, 0.006598], [0,0,0,0], [9E9, 9E9, 9E9, 9E9, 9E9, 9E9]];
	VAR robtarget Openhole_7519 := [[438.71, -10.53, 182.41], [-0.063612, 0.70424, 0.707058, 0.008284], [0,0,0,0], [9E9, 9E9, 9E9, 9E9, 9E9, 9E9]];
	VAR robtarget Openhole_7520 := [[438.21, -10.53, 182.45], [-0.06528, 0.704087, 0.707037, 0.009964], [0,0,0,0], [9E9, 9E9, 9E9, 9E9, 9E9, 9E9]];
	VAR robtarget Openhole_7521 := [[437.72, -10.53, 182.49], [-0.06694, 0.703931, 0.707011, 0.011649], [0,0,0,0], [9E9, 9E9, 9E9, 9E9, 9E9, 9E9]];
	VAR robtarget Openhole_7522 := [[437.22, -10.53, 182.53], [-0.068613, 0.70377, 0.706981, 0.013315], [0,0,0,0], [9E9, 9E9, 9E9, 9E9, 9E9, 9E9]];
	VAR robtarget Openhole_7523 := [[438.63, -8.96, 182.58], [-0.069183, 0.703714, 0.707099, 0.003295], [0,0,0,0], [9E9, 9E9, 9E9, 9E9, 9E9, 9E9]];
	VAR robtarget Openhole_7524 := [[444.58, -8.42, 182.03], [-0.050988, 0.705266, 0.706859, -0.018706], [0,0,0,0], [9E9, 9E9, 9E9, 9E9, 9E9, 9E9]];
	VAR robtarget Openhole_7525 := [[445.07, -8.4, 181.98], [-0.049394, 0.705379, 0.70681, -0.020484], [0,0,0,0], [9E9, 9E9, 9E9, 9E9, 9E9, 9E9]];
	VAR robtarget Openhole_7526 := [[446.57, -8.37, 181.83], [-0.04444, 0.705709, 0.706641, -0.025659], [0,0,0,0], [9E9, 9E9, 9E9, 9E9, 9E9, 9E9]];
	VAR robtarget Openhole_7527 := [[447.06, -8.37, 181.78], [-0.042739, 0.705814, 0.706578, -0.027339], [0,0,0,0], [9E9, 9E9, 9E9, 9E9, 9E9, 9E9]];
	VAR robtarget Openhole_7528 := [[452.53, -8.5, 181.22], [-0.023637, 0.706712, 0.705646, -0.045423], [0,0,0,0], [9E9, 9E9, 9E9, 9E9, 9E9, 9E9]];
	VAR robtarget Openhole_7529 := [[453.03, -8.5, 181.17], [-0.021943, 0.706766, 0.705536, -0.047107], [0,0,0,0], [9E9, 9E9, 9E9, 9E9, 9E9, 9E9]];
	VAR robtarget Openhole_7530 := [[453.53, -8.5, 181.12], [-0.020258, 0.706817, 0.705421, -0.048799], [0,0,0,0], [9E9, 9E9, 9E9, 9E9, 9E9, 9E9]];
	VAR robtarget Openhole_7531 := [[454.03, -8.5, 181.07], [-0.018552, 0.706863, 0.705303, -0.050469], [0,0,0,0], [9E9, 9E9, 9E9, 9E9, 9E9, 9E9]];
	VAR robtarget Openhole_7532 := [[454.52, -8.49, 181.02], [-0.016873, 0.706905, 0.70518, -0.052163], [0,0,0,0], [9E9, 9E9, 9E9, 9E9, 9E9, 9E9]];
	VAR robtarget Openhole_7533 := [[455.02, -8.48, 180.97], [-0.015215, 0.706943, 0.705051, -0.053876], [0,0,0,0], [9E9, 9E9, 9E9, 9E9, 9E9, 9E9]];
	VAR robtarget Openhole_7534 := [[457.01, -8.37, 180.76], [-0.008801, 0.707052, 0.704479, -0.060899], [0,0,0,0], [9E9, 9E9, 9E9, 9E9, 9E9, 9E9]];
	VAR robtarget Openhole_7535 := [[454.64, -6.86, 180.92], [-0.021967, 0.706765, 0.704726, -0.057982], [0,0,0,0], [9E9, 9E9, 9E9, 9E9, 9E9, 9E9]];
	VAR robtarget Openhole_7536 := [[453.65, -6.78, 181.03], [-0.025619, 0.706643, 0.704971, -0.054915], [0,0,0,0], [9E9, 9E9, 9E9, 9E9, 9E9, 9E9]];
	VAR robtarget Openhole_7537 := [[452.66, -6.67, 181.15], [-0.029382, 0.706496, 0.705194, -0.051977], [0,0,0,0], [9E9, 9E9, 9E9, 9E9, 9E9, 9E9]];
	VAR robtarget Openhole_7538 := [[449.69, -6.4, 181.5], [-0.040412, 0.705951, 0.705808, -0.042843], [0,0,0,0], [9E9, 9E9, 9E9, 9E9, 9E9, 9E9]];
	VAR robtarget Openhole_7539 := [[448.2, -6.35, 181.68], [-0.045666, 0.705631, 0.706086, -0.037982], [0,0,0,0], [9E9, 9E9, 9E9, 9E9, 9E9, 9E9]];
	VAR robtarget Openhole_7540 := [[447.71, -6.35, 181.74], [-0.047331, 0.705521, 0.706176, -0.036276], [0,0,0,0], [9E9, 9E9, 9E9, 9E9, 9E9, 9E9]];
	VAR robtarget Openhole_7541 := [[447.21, -6.37, 181.8], [-0.048966, 0.705409, 0.706263, -0.03454], [0,0,0,0], [9E9, 9E9, 9E9, 9E9, 9E9, 9E9]];
	VAR robtarget Openhole_7542 := [[446.22, -6.44, 181.92], [-0.05209, 0.705186, 0.70643, -0.030938], [0,0,0,0], [9E9, 9E9, 9E9, 9E9, 9E9, 9E9]];
	VAR robtarget Openhole_7543 := [[445.24, -6.56, 182.03], [-0.055007, 0.704964, 0.706585, -0.027169], [0,0,0,0], [9E9, 9E9, 9E9, 9E9, 9E9, 9E9]];
	VAR robtarget Openhole_7544 := [[444.74, -6.64, 182.09], [-0.056416, 0.704853, 0.706656, -0.025246], [0,0,0,0], [9E9, 9E9, 9E9, 9E9, 9E9, 9E9]];
	VAR robtarget Openhole_7545 := [[441.88, -4.7, 182.57], [-0.072526, 0.703378, 0.706766, -0.021951], [0,0,0,0], [9E9, 9E9, 9E9, 9E9, 9E9, 9E9]];
	VAR robtarget Openhole_7546 := [[439.03, -2.77, 183.16], [-0.088397, 0.70156, 0.706862, -0.018619], [0,0,0,0], [9E9, 9E9, 9E9, 9E9, 9E9, 9E9]];
	VAR robtarget Openhole_7547 := [[445.19, -0.91, 182.27], [-0.073984, 0.703226, 0.705623, -0.04578], [0,0,0,0], [9E9, 9E9, 9E9, 9E9, 9E9, 9E9]];
	VAR robtarget Openhole_7548 := [[446.14, -0.63, 182.11], [-0.071675, 0.703465, 0.705344, -0.049902], [0,0,0,0], [9E9, 9E9, 9E9, 9E9, 9E9, 9E9]];
	VAR robtarget Openhole_7549 := [[447.09, -0.38, 181.95], [-0.069285, 0.703704, 0.705044, -0.053973], [0,0,0,0], [9E9, 9E9, 9E9, 9E9, 9E9, 9E9]];
	VAR robtarget Openhole_7550 := [[447.57, -0.24, 181.86], [-0.068131, 0.703817, 0.704883, -0.05603], [0,0,0,0], [9E9, 9E9, 9E9, 9E9, 9E9, 9E9]];
	VAR robtarget Openhole_7551 := [[448.05, -0.13, 181.78], [-0.066896, 0.703935, 0.704721, -0.058038], [0,0,0,0], [9E9, 9E9, 9E9, 9E9, 9E9, 9E9]];
	VAR robtarget Openhole_7552 := [[448.52, 0, 181.69], [-0.065696, 0.704048, 0.704551, -0.060065], [0,0,0,0], [9E9, 9E9, 9E9, 9E9, 9E9, 9E9]];
	VAR robtarget Openhole_7553 := [[449.49, 0.16, 181.51], [-0.062922, 0.704302, 0.704216, -0.063876], [0,0,0,0], [9E9, 9E9, 9E9, 9E9, 9E9, 9E9]];
	VAR robtarget Openhole_7554 := [[450.48, 0.12, 181.33], [-0.059462, 0.704602, 0.703918, -0.067082], [0,0,0,0], [9E9, 9E9, 9E9, 9E9, 9E9, 9E9]];
	VAR robtarget Openhole_7555 := [[451.43, -0.1, 181.16], [-0.055439, 0.70493, 0.703677, -0.069563], [0,0,0,0], [9E9, 9E9, 9E9, 9E9, 9E9, 9E9]];
	VAR robtarget Openhole_7556 := [[451.9, -0.27, 181.08], [-0.053302, 0.705095, 0.703576, -0.070574], [0,0,0,0], [9E9, 9E9, 9E9, 9E9, 9E9, 9E9]];
	VAR robtarget Openhole_7557 := [[452.84, -0.58, 180.92], [-0.049081, 0.705401, 0.703357, -0.072721], [0,0,0,0], [9E9, 9E9, 9E9, 9E9, 9E9, 9E9]];
	VAR robtarget Openhole_7558 := [[453.8, -0.8, 180.76], [-0.045059, 0.70567, 0.703095, -0.075219], [0,0,0,0], [9E9, 9E9, 9E9, 9E9, 9E9, 9E9]];
	VAR robtarget Openhole_7559 := [[454.77, -0.99, 180.6], [-0.041107, 0.705911, 0.702811, -0.077826], [0,0,0,0], [9E9, 9E9, 9E9, 9E9, 9E9, 9E9]];
	VAR robtarget Openhole_7560 := [[457.21, -1.38, 180.21], [-0.031477, 0.706406, 0.702018, -0.084683], [0,0,0,0], [9E9, 9E9, 9E9, 9E9, 9E9, 9E9]];
	VAR robtarget Openhole_7561 := [[459.17, -1.56, 179.89], [-0.024132, 0.706695, 0.701281, -0.090582], [0,0,0,0], [9E9, 9E9, 9E9, 9E9, 9E9, 9E9]];
	VAR robtarget Openhole_7562 := [[460.16, -1.6, 179.73], [-0.020601, 0.706807, 0.700875, -0.093672], [0,0,0,0], [9E9, 9E9, 9E9, 9E9, 9E9, 9E9]];
	VAR robtarget Openhole_7563 := [[461.14, -1.61, 179.56], [-0.017177, 0.706898, 0.700442, -0.096856], [0,0,0,0], [9E9, 9E9, 9E9, 9E9, 9E9, 9E9]];
	VAR robtarget Openhole_7564 := [[461.64, -1.61, 179.48], [-0.015494, 0.706937, 0.700217, -0.09847], [0,0,0,0], [9E9, 9E9, 9E9, 9E9, 9E9, 9E9]];
	VAR robtarget Openhole_7565 := [[467.04, -1.32, 178.52], [0.002033, 0.707104, 0.697396, -0.116786], [0,0,0,0], [9E9, 9E9, 9E9, 9E9, 9E9, 9E9]];
	VAR robtarget Openhole_7566 := [[474.41, -0.89, 177.17], [0.025502, 0.706647, 0.69291, -0.14098], [0,0,0,0], [9E9, 9E9, 9E9, 9E9, 9E9, 9E9]];
	VAR robtarget Openhole_7567 := [[476.87, -0.86, 176.73], [0.033594, 0.706308, 0.691345, -0.148468], [0,0,0,0], [9E9, 9E9, 9E9, 9E9, 9E9, 9E9]];
	VAR robtarget Openhole_7568 := [[477.36, -0.86, 176.64], [0.035235, 0.706228, 0.69103, -0.149923], [0,0,0,0], [9E9, 9E9, 9E9, 9E9, 9E9, 9E9]];
	VAR robtarget Openhole_7569 := [[482.78, -1.08, 175.76], [0.053671, 0.705067, 0.687581, -0.165022], [0,0,0,0], [9E9, 9E9, 9E9, 9E9, 9E9, 9E9]];
	VAR robtarget Openhole_7570 := [[488.7, -1.64, 174.95], [0.074268, 0.703196, 0.683874, -0.179769], [0,0,0,0], [9E9, 9E9, 9E9, 9E9, 9E9, 9E9]];
	VAR robtarget Openhole_7571 := [[495.1, -2.58, 174.3], [0.096735, 0.700459, 0.679997, -0.193918], [0,0,0,0], [9E9, 9E9, 9E9, 9E9, 9E9, 9E9]];
	VAR robtarget Openhole_7572 := [[495.59, -2.66, 174.25], [0.098457, 0.700219, 0.679706, -0.194935], [0,0,0,0], [9E9, 9E9, 9E9, 9E9, 9E9, 9E9]];
	VAR robtarget Openhole_7573 := [[495.54, -3.95, 174.83], [0.102181, 0.699685, 0.680813, -0.191035], [0,0,0,0], [9E9, 9E9, 9E9, 9E9, 9E9, 9E9]];
	VAR robtarget Openhole_7574 := [[488.63, -3.04, 175.49], [0.078358, 0.702752, 0.685012, -0.175381], [0,0,0,0], [9E9, 9E9, 9E9, 9E9, 9E9, 9E9]];
	VAR robtarget Openhole_7575 := [[482.7, -2.51, 176.24], [0.057926, 0.70473, 0.68868, -0.160374], [0,0,0,0], [9E9, 9E9, 9E9, 9E9, 9E9, 9E9]];
	VAR robtarget Openhole_7576 := [[477.26, -2.32, 177.05], [0.039574, 0.705999, 0.692061, -0.145093], [0,0,0,0], [9E9, 9E9, 9E9, 9E9, 9E9, 9E9]];
	VAR robtarget Openhole_7577 := [[476.77, -2.31, 177.13], [0.037937, 0.706088, 0.692367, -0.143625], [0,0,0,0], [9E9, 9E9, 9E9, 9E9, 9E9, 9E9]];
	VAR robtarget Openhole_7578 := [[476.28, -2.32, 177.21], [0.036315, 0.706174, 0.692674, -0.142135], [0,0,0,0], [9E9, 9E9, 9E9, 9E9, 9E9, 9E9]];
	VAR robtarget Openhole_7579 := [[470.37, -2.56, 178.21], [0.017326, 0.706894, 0.696278, -0.123278], [0,0,0,0], [9E9, 9E9, 9E9, 9E9, 9E9, 9E9]];
	VAR robtarget Openhole_7580 := [[462.5, -3.12, 179.53], [-0.007548, 0.707066, 0.700513, -0.096343], [0,0,0,0], [9E9, 9E9, 9E9, 9E9, 9E9, 9E9]];
	VAR robtarget Openhole_7581 := [[461.51, -3.15, 179.68], [-0.010828, 0.707024, 0.700961, -0.093027], [0,0,0,0], [9E9, 9E9, 9E9, 9E9, 9E9, 9E9]];
	VAR robtarget Openhole_7582 := [[461.02, -3.16, 179.76], [-0.012513, 0.706996, 0.701174, -0.091406], [0,0,0,0], [9E9, 9E9, 9E9, 9E9, 9E9, 9E9]];
	VAR robtarget Openhole_7583 := [[460.52, -3.16, 179.83], [-0.014208, 0.706964, 0.701383, -0.089788], [0,0,0,0], [9E9, 9E9, 9E9, 9E9, 9E9, 9E9]];
	VAR robtarget Openhole_7584 := [[459.53, -3.13, 179.98], [-0.017681, 0.706886, 0.701781, -0.086625], [0,0,0,0], [9E9, 9E9, 9E9, 9E9, 9E9, 9E9]];
	VAR robtarget Openhole_7585 := [[458.55, -3.07, 180.13], [-0.021253, 0.706787, 0.702153, -0.083553], [0,0,0,0], [9E9, 9E9, 9E9, 9E9, 9E9, 9E9]];
	VAR robtarget Openhole_7586 := [[454.62, -2.55, 180.7], [-0.036449, 0.706167, 0.703406, -0.072253], [0,0,0,0], [9E9, 9E9, 9E9, 9E9, 9E9, 9E9]];
	VAR robtarget Openhole_7587 := [[451.22, -1.9, 181.23], [-0.050212, 0.705322, 0.704299, -0.062954], [0,0,0,0], [9E9, 9E9, 9E9, 9E9, 9E9, 9E9]];
	VAR robtarget Openhole_7588 := [[450.74, -1.83, 181.31], [-0.052108, 0.705184, 0.704425, -0.06153], [0,0,0,0], [9E9, 9E9, 9E9, 9E9, 9E9, 9E9]];
	VAR robtarget Openhole_7589 := [[450.25, -1.78, 181.39], [-0.053951, 0.705046, 0.704553, -0.060043], [0,0,0,0], [9E9, 9E9, 9E9, 9E9, 9E9, 9E9]];
